	LOCAL CONST Robtarget Tr_meulage_bavure_P268 :=[[-161.9653125,-184.567296875,19.5],[0.560964234006759,-0.570777278642454,0.427648680140188,-0.420296362969132],[0,0,0,0],[8.999999E+09,8.999999E+09,8.999999E+09,8.999999E+09,8.999999E+09,8.999999E+09]];
	LOCAL CONST Robtarget Tr_meulage_bavure_P269 :=[[-161.438453125,-185.88871875,19.5],[0.561482497351615,-0.570629960328972,0.427154440312253,-0.420306956478566],[0,0,0,0],[8.999999E+09,8.999999E+09,8.999999E+09,8.999999E+09,8.999999E+09,8.999999E+09]];
	LOCAL CONST Robtarget Tr_meulage_bavure_P270 :=[[-161.127265625,-186.709515625,19.5],[0.562125073730672,-0.570599348324866,0.426494180054633,-0.420160088007001],[0,0,0,0],[8.999999E+09,8.999999E+09,8.999999E+09,8.999999E+09,8.999999E+09,8.999999E+09]];
	LOCAL CONST Robtarget Tr_meulage_bavure_P271 :=[[-159.300578125,-195.6424375,19.5],[0.562874001364667,-0.570656851193447,0.425695264639237,-0.41988945978369],[0,0,0,0],[8.999999E+09,8.999999E+09,8.999999E+09,8.999999E+09,8.999999E+09,8.999999E+09]];
	LOCAL CONST Robtarget Tr_meulage_bavure_P272 :=[[-159.28934375,-195.682734375,19.5],[0.563712315179465,-0.570787324955456,0.424779737224237,-0.419514517304122],[0,0,0,0],[8.999999E+09,8.999999E+09,8.999999E+09,8.999999E+09,8.999999E+09,8.999999E+09]];
	LOCAL CONST Robtarget Tr_meulage_bavure_P273 :=[[-159.286125,-195.694703125,19.5],[0.564604788725629,-0.570963377966838,0.423792547953419,-0.419072940987527],[0,0,0,0],[8.999999E+09,8.999999E+09,8.999999E+09,8.999999E+09,8.999999E+09,8.999999E+09]];
	LOCAL CONST Robtarget Tr_meulage_bavure_P274 :=[[-159.284375,-195.70196875,19.5],[0.565530486147354,-0.571160305808485,0.422763052996336,-0.418595957132785],[0,0,0,0],[8.999999E+09,8.999999E+09,8.999999E+09,8.999999E+09,8.999999E+09,8.999999E+09]];
	LOCAL CONST Robtarget Tr_meulage_bavure_P275 :=[[-157.99475,-199.292578125,19.5],[0.566472293460366,-0.571359278782923,0.421714944239663,-0.418107906042624],[0,0,0,0],[8.999999E+09,8.999999E+09,8.999999E+09,8.999999E+09,8.999999E+09,8.999999E+09]];
	LOCAL CONST Robtarget Tr_meulage_bavure_P276 :=[[-157.544234375,-200.938265625,19.5],[0.567401299111796,-0.571538107883857,0.420685514492802,-0.417640581000833],[0,0,0,0],[8.999999E+09,8.999999E+09,8.999999E+09,8.999999E+09,8.999999E+09,8.999999E+09]];
	LOCAL CONST Robtarget Tr_meulage_bavure_P277 :=[[-156.8125,-202.558203125,19.5],[0.568302601605658,-0.571679624762868,0.419695994543555,-0.41721676836307],[0,0,0,0],[8.999999E+09,8.999999E+09,8.999999E+09,8.999999E+09,8.999999E+09,8.999999E+09]];
	LOCAL CONST Robtarget Tr_meulage_bavure_P278 :=[[-156.25728125,-204.908390625,19.5],[0.569171214806915,-0.571775396245421,0.418754532827547,-0.416847293046261],[0,0,0,0],[8.999999E+09,8.999999E+09,8.999999E+09,8.999999E+09,8.999999E+09,8.999999E+09]];
	LOCAL CONST Robtarget Tr_meulage_bavure_P279 :=[[-155.75175,-206.384375,19.5],[0.569996546823764,-0.57181706101586,0.417875161306644,-0.416544757382824],[0,0,0,0],[8.999999E+09,8.999999E+09,8.999999E+09,8.999999E+09,8.999999E+09,8.999999E+09]];
	LOCAL CONST Robtarget Tr_meulage_bavure_P280 :=[[-155.11828125,-208.979578125,19.5],[0.570780006509268,-0.571805632479948,0.417056295855806,-0.416308237872519],[0,0,0,0],[8.999999E+09,8.999999E+09,8.999999E+09,8.999999E+09,8.999999E+09,8.999999E+09]];
	LOCAL CONST Robtarget Tr_meulage_bavure_P281 :=[[-154.511328125,-211.640203125,19.5],[0.571520591827226,-0.571739384929797,0.4162997144144,-0.416140404930889],[0,0,0,0],[8.999999E+09,8.999999E+09,8.999999E+09,8.999999E+09,8.999999E+09,8.999999E+09]];
	LOCAL CONST Robtarget Tr_meulage_bavure_P282 :=[[-154.18290625,-212.67675,19.5],[0.572213364310843,-0.57162923861389,0.415607199226649,-0.416031892066882],[0,0,0,0],[8.999999E+09,8.999999E+09,8.999999E+09,8.999999E+09,8.999999E+09,8.999999E+09]];
	LOCAL CONST Robtarget Tr_meulage_bavure_P283 :=[[-152.8583125,-215.9785,19.5],[0.572864706832717,-0.571464182646808,0.414975670626358,-0.415992678307547],[0,0,0,0],[8.999999E+09,8.999999E+09,8.999999E+09,8.999999E+09,8.999999E+09,8.999999E+09]];
	LOCAL CONST Robtarget Tr_meulage_bavure_P284 :=[[-152.411953125,-217.957359375,19.5],[0.573480034959651,-0.571248401283081,0.4143980984857,-0.416016982232263],[0,0,0,0],[8.999999E+09,8.999999E+09,8.999999E+09,8.999999E+09,8.999999E+09,8.999999E+09]];
	LOCAL CONST Robtarget Tr_meulage_bavure_P285 :=[[-151.933640625,-219.27084375,19.5],[0.574050202363302,-0.570970854337552,0.413887624220456,-0.416119794267042],[0,0,0,0],[8.999999E+09,8.999999E+09,8.999999E+09,8.999999E+09,8.999999E+09,8.999999E+09]];
	LOCAL CONST Robtarget Tr_meulage_bavure_P286 :=[[-151.668234375,-220.093296875,19.5],[0.574574547686089,-0.570649212284852,0.413439168547303,-0.416283100282631],[0,0,0,0],[8.999999E+09,8.999999E+09,8.999999E+09,8.999999E+09,8.999999E+09,8.999999E+09]];
	LOCAL CONST Robtarget Tr_meulage_bavure_P287 :=[[-149.616609375,-228.880140625,19.5],[0.575057843902687,-0.570279616930627,0.413048830883079,-0.41650966133521],[0,0,0,0],[8.999999E+09,8.999999E+09,8.999999E+09,8.999999E+09,8.999999E+09,8.999999E+09]];
	LOCAL CONST Robtarget Tr_meulage_bavure_P288 :=[[-149.551046875,-229.11575,19.5],[0.575509045661707,-0.569878410393925,0.412701822474269,-0.416779487804835],[0,0,0,0],[8.999999E+09,8.999999E+09,8.999999E+09,8.999999E+09,8.999999E+09,8.999999E+09]];
	LOCAL CONST Robtarget Tr_meulage_bavure_P289 :=[[-147.845921875,-233.037921875,19.5],[0.575938029590918,-0.569448353003208,0.412386744830926,-0.417086480265925],[0,0,0,0],[8.999999E+09,8.999999E+09,8.999999E+09,8.999999E+09,8.999999E+09,8.999999E+09]];
	LOCAL CONST Robtarget Tr_meulage_bavure_P290 :=[[-147.505546875,-234.7584375,19.5],[0.576374910636539,-0.569018116570961,0.412062744044535,-0.417390273453091],[0,0,0,0],[8.999999E+09,8.999999E+09,8.999999E+09,8.999999E+09,8.999999E+09,8.999999E+09]];
	LOCAL CONST Robtarget Tr_meulage_bavure_P291 :=[[-146.999359375,-236.0205,19.5],[0.576853982153147,-0.568620156737828,0.411683557372683,-0.417644884099493],[0,0,0,0],[8.999999E+09,8.999999E+09,8.999999E+09,8.999999E+09,8.999999E+09,8.999999E+09]];
	LOCAL CONST Robtarget Tr_meulage_bavure_P292 :=[[-146.427,-238.509484375,19.5],[0.577416776077298,-0.568301736935537,0.41119083020271,-0.417785954356722],[0,0,0,0],[8.999999E+09,8.999999E+09,8.999999E+09,8.999999E+09,8.999999E+09,8.999999E+09]];
	LOCAL CONST Robtarget Tr_meulage_bavure_P293 :=[[-146.179640625,-239.26884375,19.5],[0.578126284754704,-0.568116391381928,0.410501698615583,-0.417734509171339],[0,0,0,0],[8.999999E+09,8.999999E+09,8.999999E+09,8.999999E+09,8.999999E+09,8.999999E+09]];
	LOCAL CONST Robtarget Tr_meulage_bavure_P294 :=[[-145.538734375,-242.18440625,19.5],[0.57903388760407,-0.568130354419907,0.409541192289515,-0.417401089134791],[0,0,0,0],[8.999999E+09,8.999999E+09,8.999999E+09,8.999999E+09,8.999999E+09,8.999999E+09]];
	LOCAL CONST Robtarget Tr_meulage_bavure_P295 :=[[-145.2123125,-243.432875,19.5],[0.580214944471463,-0.568413693302016,0.408206746970448,-0.416681824905458],[0,0,0,0],[8.999999E+09,8.999999E+09,8.999999E+09,8.999999E+09,8.999999E+09,8.999999E+09]];
	LOCAL CONST Robtarget Tr_meulage_bavure_P296 :=[[-144.365421875,-245.033828125,19.5],[0.581756623872827,-0.569033712901752,0.406381818028901,-0.415468027815452],[0,0,0,0],[8.999999E+09,8.999999E+09,8.999999E+09,8.999999E+09,8.999999E+09,8.999999E+09]];
	LOCAL CONST Robtarget Tr_meulage_bavure_P297 :=[[-144.034125,-246.257625,19.5],[0.583714280713272,-0.570060460460229,0.403978570192655,-0.413654475059025],[0,0,0,0],[8.999999E+09,8.999999E+09,8.999999E+09,8.999999E+09,8.999999E+09,8.999999E+09]];
	LOCAL CONST Robtarget Tr_meulage_bavure_P298 :=[[-143.6095,-247.7546875,19.5],[0.58617245989944,-0.571557348115518,0.400874380777533,-0.4111250125045],[0,0,0,0],[8.999999E+09,8.999999E+09,8.999999E+09,8.999999E+09,8.999999E+09,8.999999E+09]];
	LOCAL CONST Robtarget Tr_meulage_bavure_P299 :=[[-142.860328125,-249.55490625,19.5],[0.589188052385461,-0.573590439879237,0.396966412920798,-0.407761098215811],[0,0,0,0],[8.999999E+09,8.999999E+09,8.999999E+09,8.999999E+09,8.999999E+09,8.999999E+09]];
	LOCAL CONST Robtarget Tr_meulage_bavure_P300 :=[[-142.402375,-251.853640625,19.5],[0.592808671964743,-0.576208210016921,0.392156346958513,-0.403454305581994],[0,0,0,0],[8.999999E+09,8.999999E+09,8.999999E+09,8.999999E+09,8.999999E+09,8.999999E+09]];
	LOCAL CONST Robtarget Tr_meulage_bavure_P301 :=[[-140.7485625,-258.0768125,19.5],[0.597072072972443,-0.579441265135707,0.386348990807515,-0.398104530539827],[0,0,0,0],[8.999999E+09,8.999999E+09,8.999999E+09,8.999999E+09,8.999999E+09,8.999999E+09]];
	LOCAL CONST Robtarget Tr_meulage_bavure_P302 :=[[-140.3933125,-259.20978125,19.5],[0.602013083361173,-0.583316118473957,0.379437191320676,-0.391599248254036],[0,0,0,0],[8.999999E+09,8.999999E+09,8.999999E+09,8.999999E+09,8.999999E+09,8.999999E+09]];
	LOCAL CONST Robtarget Tr_meulage_bavure_P303 :=[[-140.164671875,-259.836421875,19.5],[0.607618116502847,-0.587817465101063,0.371364545167804,-0.383873972563918],[0,0,0,0],[8.999999E+09,8.999999E+09,8.999999E+09,8.999999E+09,8.999999E+09,8.999999E+09]];
	LOCAL CONST Robtarget Tr_meulage_bavure_P304 :=[[-138.449671875,-263.1504375,19.5],[0.613883056235529,-0.592942762212286,0.362039441275421,-0.374825181875461],[0,0,0,0],[8.999999E+09,8.999999E+09,8.999999E+09,8.999999E+09,8.999999E+09,8.999999E+09]];
	LOCAL CONST Robtarget Tr_meulage_bavure_P305 :=[[-137.6564375,-265.19478125,19.5],[0.620753084659352,-0.59864213211971,0.351426859012845,-0.36440687191851],[0,0,0,0],[8.999999E+09,8.999999E+09,8.999999E+09,8.999999E+09,8.999999E+09,8.999999E+09]];
	LOCAL CONST Robtarget Tr_meulage_bavure_P306 :=[[-136.8803125,-266.6085625,19.5],[0.628170166944891,-0.604841141121465,0.339490203423159,-0.35258451064534],[0,0,0,0],[8.999999E+09,8.999999E+09,8.999999E+09,8.999999E+09,8.999999E+09,8.999999E+09]];
	LOCAL CONST Robtarget Tr_meulage_bavure_P307 :=[[-134.9164375,-269.53475,19.5],[0.636031217124536,-0.611449574748402,0.326239235907522,-0.339354783873095],[0,0,0,0],[8.999999E+09,8.999999E+09,8.999999E+09,8.999999E+09,8.999999E+09,8.999999E+09]];
	LOCAL CONST Robtarget Tr_meulage_bavure_P308 :=[[-133.2449375,-272.6095625,19.5],[0.644224659383251,-0.618344665454578,0.311705957595993,-0.32475199606094],[0,0,0,0],[8.999999E+09,8.999999E+09,8.999999E+09,8.999999E+09,8.999999E+09,8.999999E+09]];
	LOCAL CONST Robtarget Tr_meulage_bavure_P309 :=[[-132.551703125,-273.5116875,19.5],[0.652594348190598,-0.625402876804148,0.29598013661176,-0.308848858061784],[0,0,0,0],[8.999999E+09,8.999999E+09,8.999999E+09,8.999999E+09,8.999999E+09,8.999999E+09]];
	LOCAL CONST Robtarget Tr_meulage_bavure_P310 :=[[-132.1574375,-273.93109375,19.5],[0.660998089293367,-0.63246286972877,0.27917792373045,-0.291773767269302],[0,0,0,0],[8.999999E+09,8.999999E+09,8.999999E+09,8.999999E+09,8.999999E+09,8.999999E+09]];
	LOCAL CONST Robtarget Tr_meulage_bavure_P311 :=[[-130.1533828125,-275.91075,19.5],[0.669271343454706,-0.639374635521518,0.261469816707866,-0.273695961301611],[0,0,0,0],[8.999999E+09,8.999999E+09,8.999999E+09,8.999999E+09,8.999999E+09,8.999999E+09]];
	LOCAL CONST Robtarget Tr_meulage_bavure_P312 :=[[-129.5635390625,-276.394625,19.5],[0.677256054189009,-0.645991723265792,0.243065647445525,-0.25482939698613],[0,0,0,0],[8.999999E+09,8.999999E+09,8.999999E+09,8.999999E+09,8.999999E+09,8.999999E+09]];
	LOCAL CONST Robtarget Tr_meulage_bavure_P313 :=[[-125.70825,-279.1965,19.5],[0.684815904495517,-0.652189819896316,0.224188779708599,-0.235403922708113],[0,0,0,0],[8.999999E+09,8.999999E+09,8.999999E+09,8.999999E+09,8.999999E+09,8.999999E+09]];
	LOCAL CONST Robtarget Tr_meulage_bavure_P314 :=[[-124.69521875,-279.913875,19.5],[0.691839849635144,-0.657856194737078,0.205091279018427,-0.215685921593087],[0,0,0,0],[8.999999E+09,8.999999E+09,8.999999E+09,8.999999E+09,8.999999E+09,8.999999E+09]];
	LOCAL CONST Robtarget Tr_meulage_bavure_P315 :=[[-119.5407109375,-282.797625,19.5],[0.698244372547129,-0.662926894954686,0.186008064006495,-0.195917656877987],[0,0,0,0],[8.999999E+09,8.999999E+09,8.999999E+09,8.999999E+09,8.999999E+09,8.999999E+09]];
	LOCAL CONST Robtarget Tr_meulage_bavure_P316 :=[[-116.7555546875,-284.14571875,19.5],[0.703994145177397,-0.667352092209407,0.167154061077636,-0.176331926901872],[0,0,0,0],[8.999999E+09,8.999999E+09,8.999999E+09,8.999999E+09,8.999999E+09,8.999999E+09]];
	LOCAL CONST Robtarget Tr_meulage_bavure_P317 :=[[-112.591765625,-285.93153125,19.5],[0.709058736177083,-0.67112758152923,0.148747698148336,-0.157154701670856],[0,0,0,0],[8.999999E+09,8.999999E+09,8.999999E+09,8.999999E+09,8.999999E+09,8.999999E+09]];
	LOCAL CONST Robtarget Tr_meulage_bavure_P318 :=[[-111.89978125,-286.17246875,19.5],[0.713459335022752,-0.674262369715255,0.130947400243534,-0.138559779244634],[0,0,0,0],[8.999999E+09,8.999999E+09,8.999999E+09,8.999999E+09,8.999999E+09,8.999999E+09]];
	LOCAL CONST Robtarget Tr_meulage_bavure_P319 :=[[-109.451328125,-286.99928125,19.5],[0.71721616316262,-0.676798706879172,0.113904788557829,-0.120707020543821],[0,0,0,0],[8.999999E+09,8.999999E+09,8.999999E+09,8.999999E+09,8.999999E+09,8.999999E+09]];
	LOCAL CONST Robtarget Tr_meulage_bavure_P320 :=[[-109.0068671875,-287.11028125,19.5],[0.720386199432233,-0.678781129299869,0.0977080074532281,-0.103696901851012],[0,0,0,0],[8.999999E+09,8.999999E+09,8.999999E+09,8.999999E+09,8.999999E+09,8.999999E+09]];
	LOCAL CONST Robtarget Tr_meulage_bavure_P321 :=[[-107.78265625,-287.435875,19.5],[0.723031240066771,-0.680253807562518,0.0824577376474849,-0.0876430526982125],[0,0,0,0],[8.999999E+09,8.999999E+09,8.999999E+09,8.999999E+09,8.999999E+09,8.999999E+09]];
	LOCAL CONST Robtarget Tr_meulage_bavure_P322 :=[[-106.4644453125,-287.84596875,19.5],[0.7252109507937,-0.681285287306183,0.0681925909536574,-0.0725892876949244],[0,0,0,0],[8.999999E+09,8.999999E+09,8.999999E+09,8.999999E+09,8.999999E+09,8.999999E+09]];
	LOCAL CONST Robtarget Tr_meulage_bavure_P323 :=[[-105.98046875,-287.92040625,19.5],[0.726986745083191,-0.681934622504451,0.0549682733471719,-0.0585997613330488],[0,0,0,0],[8.999999E+09,8.999999E+09,8.999999E+09,8.999999E+09,8.999999E+09,8.999999E+09]];
	LOCAL CONST Robtarget Tr_meulage_bavure_P324 :=[[-105.7509140625,-287.94509375,19.5],[0.728412623159497,-0.682271282005315,0.0428061076178847,-0.0457010429129395],[0,0,0,0],[8.999999E+09,8.999999E+09,8.999999E+09,8.999999E+09,8.999999E+09,8.999999E+09]];
	LOCAL CONST Robtarget Tr_meulage_bavure_P325 :=[[-103.7956875,-287.85703125,19.5],[0.729555020391346,-0.682343993654236,0.0317183960258636,-0.0339129753828471],[0,0,0,0],[8.999999E+09,8.999999E+09,8.999999E+09,8.999999E+09,8.999999E+09,8.999999E+09]];
	LOCAL CONST Robtarget Tr_meulage_bavure_P326 :=[[-98.836609375,-287.8770625,19.5],[0.730465389526081,-0.682208988231543,0.0217049125177494,-0.0232402205928225],[0,0,0,0],[8.999999E+09,8.999999E+09,8.999999E+09,8.999999E+09,8.999999E+09,8.999999E+09]];
	LOCAL CONST Robtarget Tr_meulage_bavure_P327 :=[[-98.1267734375,-287.92809375,19.5],[0.731193592992967,-0.681913551506533,0.0127567102372147,-0.013678603061212],[0,0,0,0],[8.999999E+09,8.999999E+09,8.999999E+09,8.999999E+09,8.999999E+09,8.999999E+09]];
	LOCAL CONST Robtarget Tr_meulage_bavure_P328 :=[[-96.89046875,-287.7645625,19.5],[0.731783571389712,-0.681499822687102,0.00485727743171576,-0.00521566654587902],[0,0,0,0],[8.999999E+09,8.999999E+09,8.999999E+09,8.999999E+09,8.999999E+09,8.999999E+09]];
	LOCAL CONST Robtarget Tr_meulage_bavure_P329 :=[[-95.0238984375,-287.6898125,19.5],[0.732277533985066,-0.680999874855432,-0.00201830542058397,0.00217027898357202],[0,0,0,0],[8.999999E+09,8.999999E+09,8.999999E+09,8.999999E+09,8.999999E+09,8.999999E+09]];
	LOCAL CONST Robtarget Tr_meulage_bavure_P330 :=[[-91.72903125,-287.34909375,19.5],[0.732701770281004,-0.680451088617369,-0.0078900027828738,0.00849586267586157],[0,0,0,0],[8.999999E+09,8.999999E+09,8.999999E+09,8.999999E+09,8.999999E+09,8.999999E+09]];
	LOCAL CONST Robtarget Tr_meulage_bavure_P331 :=[[-89.856875,-287.0336875,19.5],[0.733088866138208,-0.679871664260582,-0.0128162700320661,0.0138194682317681],[0,0,0,0],[8.999999E+09,8.999999E+09,8.999999E+09,8.999999E+09,8.999999E+09,8.999999E+09]];
	LOCAL CONST Robtarget Tr_meulage_bavure_P332 :=[[-85.5172734375,-286.69559375,19.5],[0.733453444169888,-0.67928812631057,-0.0168329671656543,0.0181752002795984],[0,0,0,0],[8.999999E+09,8.999999E+09,8.999999E+09,8.999999E+09,8.999999E+09,8.999999E+09]];
	LOCAL CONST Robtarget Tr_meulage_bavure_P333 :=[[-84.53634375,-286.54434375,19.5],[0.733821815164145,-0.678703060287681,-0.0200010590824421,0.0216253827923831],[0,0,0,0],[8.999999E+09,8.999999E+09,8.999999E+09,8.999999E+09,8.999999E+09,8.999999E+09]];
	LOCAL CONST Robtarget Tr_meulage_bavure_P334 :=[[-83.2665078125,-286.44875,19.5],[0.734198119116665,-0.678132647710818,-0.0223929803954049,0.0242443482749612],[0,0,0,0],[8.999999E+09,8.999999E+09,8.999999E+09,8.999999E+09,8.999999E+09,8.999999E+09]];
	LOCAL CONST Robtarget Tr_meulage_bavure_P335 :=[[-79.6076640625,-285.996375,19.5],[0.734583912009596,-0.677588173949316,-0.0240742626965029,0.0260992838279178],[0,0,0,0],[8.999999E+09,8.999999E+09,8.999999E+09,8.999999E+09,8.999999E+09,8.999999E+09]];
	LOCAL CONST Robtarget Tr_meulage_bavure_P336 :=[[-78.2538125,-285.63596875,19.5],[0.734986132932684,-0.67706581152781,-0.0251443204817685,0.0272953183596925],[0,0,0,0],[8.999999E+09,8.999999E+09,8.999999E+09,8.999999E+09,8.999999E+09,8.999999E+09]];
	LOCAL CONST Robtarget Tr_meulage_bavure_P337 :=[[-76.3402109375,-285.37465625,19.5],[0.735402485292143,-0.676567290093219,-0.0256914156380045,0.0279255754564468],[0,0,0,0],[8.999999E+09,8.999999E+09,8.999999E+09,8.999999E+09,8.999999E+09,8.999999E+09]];
	LOCAL CONST Robtarget Tr_meulage_bavure_P338 :=[[-72.4418359375,-285.24371875,19.5],[0.735825551022483,-0.67609503373989,-0.0258192860533249,0.0281003253079716],[0,0,0,0],[8.999999E+09,8.999999E+09,8.999999E+09,8.999999E+09,8.999999E+09,8.999999E+09]];
	LOCAL CONST Robtarget Tr_meulage_bavure_P339 :=[[-68.4656953125,-284.83971875,19.5],[0.736267597026046,-0.675628090950229,-0.0256273793944011,0.0279275081920483],[0,0,0,0],[8.999999E+09,8.999999E+09,8.999999E+09,8.999999E+09,8.999999E+09,8.999999E+09]];
	LOCAL CONST Robtarget Tr_meulage_bavure_P340 :=[[-65.6481015625,-284.45584375,19.5],[0.736706993967259,-0.675179101732153,-0.0252442696560809,0.0275447358567801],[0,0,0,0],[8.999999E+09,8.999999E+09,8.999999E+09,8.999999E+09,8.999999E+09,8.999999E+09]];
	LOCAL CONST Robtarget Tr_meulage_bavure_P341 :=[[-64.50961328125,-284.47453125,19.5],[0.737145027213847,-0.674739001078387,-0.0247574912343207,0.0270472901677574],[0,0,0,0],[8.999999E+09,8.999999E+09,8.999999E+09,8.999999E+09,8.999999E+09,8.999999E+09]];
	LOCAL CONST Robtarget Tr_meulage_bavure_P342 :=[[-63.09558203125,-284.451,19.5],[0.737574727550139,-0.674306700194866,-0.0242719686569887,0.0265493293542989],[0,0,0,0],[8.999999E+09,8.999999E+09,8.999999E+09,8.999999E+09,8.999999E+09,8.999999E+09]];
	LOCAL CONST Robtarget Tr_meulage_bavure_P343 :=[[-60.75375390625,-284.1825,19.5],[0.737995519441899,-0.673876223593398,-0.0238729311077847,0.0261444395523303],[0,0,0,0],[8.999999E+09,8.999999E+09,8.999999E+09,8.999999E+09,8.999999E+09,8.999999E+09]];
	LOCAL CONST Robtarget Tr_meulage_bavure_P344 :=[[-56.9111328125,-283.74796875,19.5],[0.738407827244645,-0.673441766800905,-0.0236337028553787,0.0259136157504544],[0,0,0,0],[8.999999E+09,8.999999E+09,8.999999E+09,8.999999E+09,8.999999E+09,8.999999E+09]];
	LOCAL CONST Robtarget Tr_meulage_bavure_P345 :=[[-55.53506640625,-283.48496875,19.5],[0.738803521845753,-0.673007813207025,-0.0236162827783587,0.0259250970748975],[0,0,0,0],[8.999999E+09,8.999999E+09,8.999999E+09,8.999999E+09,8.999999E+09,8.999999E+09]];
	LOCAL CONST Robtarget Tr_meulage_bavure_P346 :=[[-53.50186328125,-283.17409375,19.5],[0.739190986070497,-0.672563047793711,-0.0238471875011445,0.0262096261485151],[0,0,0,0],[8.999999E+09,8.999999E+09,8.999999E+09,8.999999E+09,8.999999E+09,8.999999E+09]];
	LOCAL CONST Robtarget Tr_meulage_bavure_P347 :=[[-49.17727734375,-282.77846875,19.5],[0.739554654010651,-0.672122706016185,-0.0243425371632662,0.0267847470236889],[0,0,0,0],[8.999999E+09,8.999999E+09,8.999999E+09,8.999999E+09,8.999999E+09,8.999999E+09]];
	LOCAL CONST Robtarget Tr_meulage_bavure_P348 :=[[-44.38299609375,-282.44271875,19.5],[0.739908728288621,-0.671670717382305,-0.0250908871651308,0.0276399818148069],[0,0,0,0],[8.999999E+09,8.999999E+09,8.999999E+09,8.999999E+09,8.999999E+09,8.999999E+09]];
	LOCAL CONST Robtarget Tr_meulage_bavure_P349 :=[[-41.2405390625,-282.2865,19.5],[0.740250211472266,-0.671209902210246,-0.0260751504918529,0.0287572272134317],[0,0,0,0],[8.999999E+09,8.999999E+09,8.999999E+09,8.999999E+09,8.999999E+09,8.999999E+09]];
	LOCAL CONST Robtarget Tr_meulage_bavure_P350 :=[[-37.7456953125,-282.0811875,19.5],[0.740566887367051,-0.670755399045768,-0.0272511663274277,0.0300874379139331],[0,0,0,0],[8.999999E+09,8.999999E+09,8.999999E+09,8.999999E+09,8.999999E+09,8.999999E+09]];
	LOCAL CONST Robtarget Tr_meulage_bavure_P351 :=[[-35.7432265625,-281.81509375,19.5],[0.740869701006427,-0.670297395744423,-0.0285705731810239,0.0315786278517456],[0,0,0,0],[8.999999E+09,8.999999E+09,8.999999E+09,8.999999E+09,8.999999E+09,8.999999E+09]];
	LOCAL CONST Robtarget Tr_meulage_bavure_P352 :=[[-32.817078125,-281.2908125,19.5],[0.741163425883474,-0.669833608837101,-0.0299837116955564,0.0331766429569906],[0,0,0,0],[8.999999E+09,8.999999E+09,8.999999E+09,8.999999E+09,8.999999E+09,8.999999E+09]];
	LOCAL CONST Robtarget Tr_meulage_bavure_P353 :=[[-31.189666015625,-281.02409375,19.5],[0.741439666191449,-0.669378732229863,-0.0314264722459313,0.0348096405961052],[0,0,0,0],[8.999999E+09,8.999999E+09,8.999999E+09,8.999999E+09,8.999999E+09,8.999999E+09]];
	LOCAL CONST Robtarget Tr_meulage_bavure_P354 :=[[-28.535064453125,-280.90421875,19.5],[0.741714526644082,-0.668919898476124,-0.0328488839806384,0.0364236353081897],[0,0,0,0],[8.999999E+09,8.999999E+09,8.999999E+09,8.999999E+09,8.999999E+09,8.999999E+09]];
	LOCAL CONST Robtarget Tr_meulage_bavure_P355 :=[[-23.35043359375,-280.3699375,19.5],[0.741979260892866,-0.668474452748739,-0.0341871288687678,0.0379463126912225],[0,0,0,0],[8.999999E+09,8.999999E+09,8.999999E+09,8.999999E+09,8.999999E+09,8.999999E+09]];
	LOCAL CONST Robtarget Tr_meulage_bavure_P356 :=[[-21.707732421875,-280.1441875,19.5],[0.742239132342601,-0.668041110268359,-0.0354126033921952,0.0393458121241323],[0,0,0,0],[8.999999E+09,8.999999E+09,8.999999E+09,8.999999E+09,8.999999E+09,8.999999E+09]];
	LOCAL CONST Robtarget Tr_meulage_bavure_P357 :=[[-18.087798828125,-279.7083125,19.5],[0.742510743010949,-0.667607685693368,-0.0364850387971614,0.0405785221569577],[0,0,0,0],[8.999999E+09,8.999999E+09,8.999999E+09,8.999999E+09,8.999999E+09,8.999999E+09]];
	LOCAL CONST Robtarget Tr_meulage_bavure_P358 :=[[-17.23358203125,-279.54203125,19.5],[0.742787417657644,-0.667185113955726,-0.0373904077498098,0.0416273142741171],[0,0,0,0],[8.999999E+09,8.999999E+09,8.999999E+09,8.999999E+09,8.999999E+09,8.999999E+09]];
	LOCAL CONST Robtarget Tr_meulage_bavure_P359 :=[[-15.7358095703125,-279.48275,19.5],[0.743060843326873,-0.666786518977901,-0.038111731974697,0.0424713681152043],[0,0,0,0],[8.999999E+09,8.999999E+09,8.999999E+09,8.999999E+09,8.999999E+09,8.999999E+09]];
	LOCAL CONST Robtarget Tr_meulage_bavure_P360 :=[[-11.11053515625,-278.86453125,19.5],[0.74334126114516,-0.66640177114528,-0.0386497263769758,0.0431120347993692],[0,0,0,0],[8.999999E+09,8.999999E+09,8.999999E+09,8.999999E+09,8.999999E+09,8.999999E+09]];
	LOCAL CONST Robtarget Tr_meulage_bavure_P361 :=[[-9.1521298828125,-278.51259375,19.5],[0.743625034281882,-0.666035033451219,-0.0390121073460656,0.0435568374118436],[0,0,0,0],[8.999999E+09,8.999999E+09,8.999999E+09,8.999999E+09,8.999999E+09,8.999999E+09]];
	LOCAL CONST Robtarget Tr_meulage_bavure_P362 :=[[-4.1391904296875,-278.02171875,19.5],[0.743913750798036,-0.665683653011691,-0.0392109822866391,0.043818995364179],[0,0,0,0],[8.999999E+09,8.999999E+09,8.999999E+09,8.999999E+09,8.999999E+09,8.999999E+09]];
	LOCAL CONST Robtarget Tr_meulage_bavure_P363 :=[[3.73715209960938,-277.50453125,19.5],[0.744208876706379,-0.665343612809414,-0.0392671951058527,0.0439216588218871],[0,0,0,0],[8.999999E+09,8.999999E+09,8.999999E+09,8.999999E+09,8.999999E+09,8.999999E+09]];
	LOCAL CONST Robtarget Tr_meulage_bavure_P364 :=[[4.41998291015625,-277.3703125,19.5],[0.744509424422736,-0.665014123771272,-0.0391961306942008,0.0438816074119574],[0,0,0,0],[8.999999E+09,8.999999E+09,8.999999E+09,8.999999E+09,8.999999E+09,8.999999E+09]];
	LOCAL CONST Robtarget Tr_meulage_bavure_P365 :=[[6.283447265625,-277.18909375,19.5],[0.744804935293087,-0.664703307286453,-0.0390252875238091,0.0437281211487018],[0,0,0,0],[8.999999E+09,8.999999E+09,8.999999E+09,8.999999E+09,8.999999E+09,8.999999E+09]];
	LOCAL CONST Robtarget Tr_meulage_bavure_P366 :=[[14.9065546875,-276.00421875,19.5],[0.745101806435219,-0.664401693705879,-0.0387708064935192,0.0434800185323727],[0,0,0,0],[8.999999E+09,8.999999E+09,8.999999E+09,8.999999E+09,8.999999E+09,8.999999E+09]];
	LOCAL CONST Robtarget Tr_meulage_bavure_P367 :=[[17.427978515625,-275.71321875,19.5],[0.745395572448328,-0.664111310053286,-0.0384543515048626,0.0431609926215477],[0,0,0,0],[8.999999E+09,8.999999E+09,8.999999E+09,8.999999E+09,8.999999E+09,8.999999E+09]];
	LOCAL CONST Robtarget Tr_meulage_bavure_P368 :=[[22.690033203125,-274.89740625,19.5],[0.745689508202804,-0.663825992976087,-0.0380935305284928,0.0427912530483325],[0,0,0,0],[8.999999E+09,8.999999E+09,8.999999E+09,8.999999E+09,8.999999E+09,8.999999E+09]];
	LOCAL CONST Robtarget Tr_meulage_bavure_P369 :=[[24.436462890625,-274.65103125,19.5],[0.745982896599928,-0.663544527508919,-0.0377029252851454,0.0423871138235338],[0,0,0,0],[8.999999E+09,8.999999E+09,8.999999E+09,8.999999E+09,8.999999E+09,8.999999E+09]];
	LOCAL CONST Robtarget Tr_meulage_bavure_P370 :=[[27.416291015625,-274.272,19.5],[0.746268856927678,-0.663272002159742,-0.0373028883472666,0.0419706903900203],[0,0,0,0],[8.999999E+09,8.999999E+09,8.999999E+09,8.999999E+09,8.999999E+09,8.999999E+09]];
	LOCAL CONST Robtarget Tr_meulage_bavure_P371 :=[[28.458375,-274.05478125,19.5],[0.746550366383039,-0.663004858448019,-0.0368947035688752,0.0415438199524097],[0,0,0,0],[8.999999E+09,8.999999E+09,8.999999E+09,8.999999E+09,8.999999E+09,8.999999E+09]];
	LOCAL CONST Robtarget Tr_meulage_bavure_P372 :=[[30.38855078125,-273.92025,19.5],[0.746830255296542,-0.662736357267652,-0.0365063043339479,0.0411385497214313],[0,0,0,0],[8.999999E+09,8.999999E+09,8.999999E+09,8.999999E+09,8.999999E+09,8.999999E+09]];
	LOCAL CONST Robtarget Tr_meulage_bavure_P373 :=[[33.11441015625,-273.5259375,19.5],[0.747099570603815,-0.662477919835629,-0.0361281719578439,0.0407430058395047],[0,0,0,0],[8.999999E+09,8.999999E+09,8.999999E+09,8.999999E+09,8.999999E+09,8.999999E+09]];
	LOCAL CONST Robtarget Tr_meulage_bavure_P374 :=[[34.83148046875,-273.24446875,19.5],[0.747355157433442,-0.662229707584567,-0.0357885259274169,0.0403889150886211],[0,0,0,0],[8.999999E+09,8.999999E+09,8.999999E+09,8.999999E+09,8.999999E+09,8.999999E+09]];
	LOCAL CONST Robtarget Tr_meulage_bavure_P375 :=[[38.11590625,-272.91428125,19.5],[0.747610535984406,-0.66197542874325,-0.0354960931727873,0.0400879731935678],[0,0,0,0],[8.999999E+09,8.999999E+09,8.999999E+09,8.999999E+09,8.999999E+09,8.999999E+09]];
	LOCAL CONST Robtarget Tr_meulage_bavure_P376 :=[[39.43502734375,-272.83925,19.5],[0.747850297504655,-0.661731773858748,-0.0352587508784534,0.0398473647114343],[0,0,0,0],[8.999999E+09,8.999999E+09,8.999999E+09,8.999999E+09,8.999999E+09,8.999999E+09]];
	LOCAL CONST Robtarget Tr_meulage_bavure_P377 :=[[45.2320859375,-272.17715625,19.5],[0.748080186236866,-0.661490302975661,-0.0350933746847424,0.0396871400105893],[0,0,0,0],[8.999999E+09,8.999999E+09,8.999999E+09,8.999999E+09,8.999999E+09,8.999999E+09]];
	LOCAL CONST Robtarget Tr_meulage_bavure_P378 :=[[47.62060546875,-271.8248125,19.5],[0.748297266506116,-0.661254439010767,-0.0350002595066617,0.0396074445337873],[0,0,0,0],[8.999999E+09,8.999999E+09,8.999999E+09,8.999999E+09,8.999999E+09,8.999999E+09]];
	LOCAL CONST Robtarget Tr_meulage_bavure_P379 :=[[48.34982421875,-271.83715625,19.5],[0.748503119203697,-0.661021600007927,-0.0349864096413146,0.039616612749036],[0,0,0,0],[8.999999E+09,8.999999E+09,8.999999E+09,8.999999E+09,8.999999E+09,8.999999E+09]];
	LOCAL CONST Robtarget Tr_meulage_bavure_P380 :=[[52.699859375,-271.37153125,19.5],[0.748708790454047,-0.660778572494331,-0.0350569386395885,0.0397219873925214],[0,0,0,0],[8.999999E+09,8.999999E+09,8.999999E+09,8.999999E+09,8.999999E+09,8.999999E+09]];
	LOCAL CONST Robtarget Tr_meulage_bavure_P381 :=[[54.4260546875,-271.0833125,19.5],[0.748899486297266,-0.660541882838812,-0.0352139747839537,0.0399243837693531],[0,0,0,0],[8.999999E+09,8.999999E+09,8.999999E+09,8.999999E+09,8.999999E+09,8.999999E+09]];
	LOCAL CONST Robtarget Tr_meulage_bavure_P382 :=[[55.685546875,-271.07,19.5],[0.749080580145308,-0.660306485593583,-0.0354475195835911,0.0402132178219008],[0,0,0,0],[8.999999E+09,8.999999E+09,8.999999E+09,8.999999E+09,8.999999E+09,8.999999E+09]];
	LOCAL CONST Robtarget Tr_meulage_bavure_P383 :=[[61.25250390625,-270.677625,19.5],[0.749249993862185,-0.660071830983981,-0.0357795012722655,0.0406134451589521],[0,0,0,0],[8.999999E+09,8.999999E+09,8.999999E+09,8.999999E+09,8.999999E+09,8.999999E+09]];
	LOCAL CONST Robtarget Tr_meulage_bavure_P384 :=[[61.646484375,-270.614125,19.5],[0.749411887250001,-0.659833714763356,-0.0362027313846949,0.0411175674167231],[0,0,0,0],[8.999999E+09,8.999999E+09,8.999999E+09,8.999999E+09,8.999999E+09,8.999999E+09]];
	LOCAL CONST Robtarget Tr_meulage_bavure_P385 :=[[61.9664296875,-270.596875,19.5],[0.749555868186807,-0.659601425194716,-0.036734234496255,0.0417439380484813],[0,0,0,0],[8.999999E+09,8.999999E+09,8.999999E+09,8.999999E+09,8.999999E+09,8.999999E+09]];
	LOCAL CONST Robtarget Tr_meulage_bavure_P386 :=[[67.4912421875,-269.82709375,19.5],[0.749684084891055,-0.659367738775831,-0.0374058686854177,0.0425295063526245],[0,0,0,0],[8.999999E+09,8.999999E+09,8.999999E+09,8.999999E+09,8.999999E+09,8.999999E+09]];
	LOCAL CONST Robtarget Tr_meulage_bavure_P387 :=[[69.15759375,-269.49821875,19.5],[0.749800250470714,-0.659124792175536,-0.0382370814766123,0.0434973370881756],[0,0,0,0],[8.999999E+09,8.999999E+09,8.999999E+09,8.999999E+09,8.999999E+09,8.999999E+09]];
	LOCAL CONST Robtarget Tr_meulage_bavure_P388 :=[[72.301265625,-268.82734375,19.5],[0.74988567242769,-0.658884441579498,-0.0392872343814879,0.0447133553516025],[0,0,0,0],[8.999999E+09,8.999999E+09,8.999999E+09,8.999999E+09,8.999999E+09,8.999999E+09]];
	LOCAL CONST Robtarget Tr_meulage_bavure_P389 :=[[209.292484375,-254.7383125,19.5],[0.749950261226932,-0.658625066039587,-0.0406112121990249,0.0462423778987642],[0,0,0,0],[8.999999E+09,8.999999E+09,8.999999E+09,8.999999E+09,8.999999E+09,8.999999E+09]];
	LOCAL CONST Robtarget Tr_meulage_bavure_P390 :=[[209.595640625,-254.598515625,19.5],[0.749979833975741,-0.658348824535315,-0.0422781521533605,0.0481625550940398],[0,0,0,0],[8.999999E+09,8.999999E+09,8.999999E+09,8.999999E+09,8.999999E+09,8.999999E+09]];
	LOCAL CONST Robtarget Tr_meulage_bavure_P391 :=[[218.53028125,-253.023828125,19.5],[0.749965349966833,-0.658047486126157,-0.0443684725768967,0.050565981582136],[0,0,0,0],[8.999999E+09,8.999999E+09,8.999999E+09,8.999999E+09,8.999999E+09,8.999999E+09]];
	LOCAL CONST Robtarget Tr_meulage_bavure_P392 :=[[219.095953125,-252.89653125,19.5],[0.749898043744128,-0.657704851819652,-0.0469840791912529,0.0535700306530519],[0,0,0,0],[8.999999E+09,8.999999E+09,8.999999E+09,8.999999E+09,8.999999E+09,8.999999E+09]];
	LOCAL CONST Robtarget Tr_meulage_bavure_P393 :=[[219.305234375,-252.853046875,19.5],[0.749762700654114,-0.657311062331293,-0.0501966798417859,0.0572569068114641],[0,0,0,0],[8.999999E+09,8.999999E+09,8.999999E+09,8.999999E+09,8.999999E+09,8.999999E+09]];
	LOCAL CONST Robtarget Tr_meulage_bavure_P394 :=[[219.690984375,-252.8630625,19.5],[0.749535210602135,-0.656855944291842,-0.0540977190566767,0.0617306512921282],[0,0,0,0],[8.999999E+09,8.999999E+09,8.999999E+09,8.999999E+09,8.999999E+09,8.999999E+09]];
	LOCAL CONST Robtarget Tr_meulage_bavure_P395 :=[[228.460390625,-252.180765625,19.5],[0.749188135675054,-0.656324703232434,-0.0587724428571624,0.0670881602907343],[0,0,0,0],[8.999999E+09,8.999999E+09,8.999999E+09,8.999999E+09,8.999999E+09,8.999999E+09]];
	LOCAL CONST Robtarget Tr_meulage_bavure_P396 :=[[229.2111875,-252.066453125,19.5],[0.748708072452323,-0.655680154651966,-0.0642809169024341,0.0734010951041143],[0,0,0,0],[8.999999E+09,8.999999E+09,8.999999E+09,8.999999E+09,8.999999E+09,8.999999E+09]];
	LOCAL CONST Robtarget Tr_meulage_bavure_P397 :=[[229.5289375,-252.008765625,19.5],[0.74806056809837,-0.654896048548644,-0.0706885228860066,0.0807445650425435],[0,0,0,0],[8.999999E+09,8.999999E+09,8.999999E+09,8.999999E+09,8.999999E+09,8.999999E+09]];
	LOCAL CONST Robtarget Tr_meulage_bavure_P398 :=[[230.121515625,-252.01496875,19.5],[0.747208688928678,-0.65394084858474,-0.0780370547917106,0.089167033264498],[0,0,0,0],[8.999999E+09,8.999999E+09,8.999999E+09,8.999999E+09,8.999999E+09,8.999999E+09]];
	LOCAL CONST Robtarget Tr_meulage_bavure_P399 :=[[236.2184375,-251.14521875,19.5],[0.746117745514469,-0.652768281572659,-0.0863604401454113,0.0987104593190307],[0,0,0,0],[8.999999E+09,8.999999E+09,8.999999E+09,8.999999E+09,8.999999E+09,8.999999E+09]];
	LOCAL CONST Robtarget Tr_meulage_bavure_P400 :=[[238.810796875,-250.59940625,19.5],[0.744722782324835,-0.651364765352148,-0.0956580684945637,0.109368431807295],[0,0,0,0],[8.999999E+09,8.999999E+09,8.999999E+09,8.999999E+09,8.999999E+09,8.999999E+09]];
	LOCAL CONST Robtarget Tr_meulage_bavure_P401 :=[[239.35559375,-250.46771875,19.5],[0.742983687419268,-0.649671188928834,-0.105940978225713,0.12115731772056],[0,0,0,0],[8.999999E+09,8.999999E+09,8.999999E+09,8.999999E+09,8.999999E+09,8.999999E+09]];
	LOCAL CONST Robtarget Tr_meulage_bavure_P402 :=[[239.716,-250.348359375,19.5],[0.740855170887779,-0.647644140892055,-0.117164267563178,0.134026926188045],[0,0,0,0],[8.999999E+09,8.999999E+09,8.999999E+09,8.999999E+09,8.999999E+09,8.999999E+09]];
	LOCAL CONST Robtarget Tr_meulage_bavure_P403 :=[[241.07934375,-250.016328125,19.5],[0.738280265150873,-0.64524724280864,-0.129287782215408,0.14792875010094],[0,0,0,0],[8.999999E+09,8.999999E+09,8.999999E+09,8.999999E+09,8.999999E+09,8.999999E+09]];
	LOCAL CONST Robtarget Tr_meulage_bavure_P404 :=[[242.75121875,-249.450046875,19.5],[0.735211311086142,-0.642438716951977,-0.142250856881771,0.162792864488882],[0,0,0,0],[8.999999E+09,8.999999E+09,8.999999E+09,8.999999E+09,8.999999E+09,8.999999E+09]];
	LOCAL CONST Robtarget Tr_meulage_bavure_P405 :=[[243.32434375,-249.18409375,19.5],[0.731621118403904,-0.639170970187056,-0.155958268975862,0.178516185018642],[0,0,0,0],[8.999999E+09,8.999999E+09,8.999999E+09,8.999999E+09,8.999999E+09,8.999999E+09]];
	LOCAL CONST Robtarget Tr_meulage_bavure_P406 :=[[245.67559375,-248.14575,19.5],[0.727468367521003,-0.635426308955196,-0.170310835968523,0.194980510040378],[0,0,0,0],[8.999999E+09,8.999999E+09,8.999999E+09,8.999999E+09,8.999999E+09,8.999999E+09]];
	LOCAL CONST Robtarget Tr_meulage_bavure_P407 :=[[247.46203125,-247.164203125,19.5],[0.722730926996024,-0.631180073813323,-0.185202431405251,0.212065511071603],[0,0,0,0],[8.999999E+09,8.999999E+09,8.999999E+09,8.999999E+09,8.999999E+09,8.999999E+09]];
	LOCAL CONST Robtarget Tr_meulage_bavure_P408 :=[[248.314765625,-246.66059375,19.5],[0.717389226773837,-0.626427510399991,-0.200519874230862,0.229636781812811],[0,0,0,0],[8.999999E+09,8.999999E+09,8.999999E+09,8.999999E+09,8.999999E+09,8.999999E+09]];
	LOCAL CONST Robtarget Tr_meulage_bavure_P409 :=[[249.07928125,-246.065078125,19.5],[0.711443692817404,-0.621171372251387,-0.216136121649987,0.247546309129759],[0,0,0,0],[8.999999E+09,8.999999E+09,8.999999E+09,8.999999E+09,8.999999E+09,8.999999E+09]];
	LOCAL CONST Robtarget Tr_meulage_bavure_P410 :=[[250.705390625,-244.898109375,19.5],[0.704909523264806,-0.615400954640711,-0.23194447789707,0.265680236771462],[0,0,0,0],[8.999999E+09,8.999999E+09,8.999999E+09,8.999999E+09,8.999999E+09,8.999999E+09]];
	LOCAL CONST Robtarget Tr_meulage_bavure_P411 :=[[252.961421875,-242.688328125,19.5],[0.697810666434406,-0.609150201754592,-0.247809719397606,0.283877876004435],[0,0,0,0],[8.999999E+09,8.999999E+09,8.999999E+09,8.999999E+09,8.999999E+09,8.999999E+09]];
	LOCAL CONST Robtarget Tr_meulage_bavure_P412 :=[[252.97034375,-242.6775625,19.5],[0.690175426010377,-0.602438874924228,-0.263634971066927,0.30202961004174],[0,0,0,0],[8.999999E+09,8.999999E+09,8.999999E+09,8.999999E+09,8.999999E+09,8.999999E+09]];
	LOCAL CONST Robtarget Tr_meulage_bavure_P413 :=[[252.9741875,-242.67371875,19.5],[0.68203699996809,-0.59529928452741,-0.279330073684175,0.320029689952783],[0,0,0,0],[8.999999E+09,8.999999E+09,8.999999E+09,8.999999E+09,8.999999E+09,8.999999E+09]];
	LOCAL CONST Robtarget Tr_meulage_bavure_P414 :=[[253.121828125,-242.486421875,19.5],[0.673442887212124,-0.587778927358809,-0.294798965257567,0.337763497582842],[0,0,0,0],[8.999999E+09,8.999999E+09,8.999999E+09,8.999999E+09,8.999999E+09,8.999999E+09]];
	LOCAL CONST Robtarget Tr_meulage_bavure_P415 :=[[256.936765625,-237.625578125,19.5],[0.664444277190496,-0.579915155410377,-0.309968715605778,0.355150123722154],[0,0,0,0],[8.999999E+09,8.999999E+09,8.999999E+09,8.999999E+09,8.999999E+09,8.999999E+09]];
	LOCAL CONST Robtarget Tr_meulage_bavure_P416 :=[[257.0650625,-237.44225,19.5],[0.655098546834546,-0.571760132361724,-0.324767698241302,0.372105075423618],[0,0,0,0],[8.999999E+09,8.999999E+09,8.999999E+09,8.999999E+09,8.999999E+09,8.999999E+09]];
	LOCAL CONST Robtarget Tr_meulage_bavure_P417 :=[[258.070796875,-235.771359375,19.5],[0.645473621108132,-0.563366986831293,-0.339127917112701,0.388553340529954],[0,0,0,0],[8.999999E+09,8.999999E+09,8.999999E+09,8.999999E+09,8.999999E+09,8.999999E+09]];
	LOCAL CONST Robtarget Tr_meulage_bavure_P418 :=[[258.29534375,-235.445703125,19.5],[0.63564962762985,-0.554806771591956,-0.352975995856972,0.404409376051697],[0,0,0,0],[8.999999E+09,8.999999E+09,8.999999E+09,8.999999E+09,8.999999E+09,8.999999E+09]];
	LOCAL CONST Robtarget Tr_meulage_bavure_P419 :=[[259.848578125,-232.276421875,19.5],[0.625694415013696,-0.546145633074355,-0.366268591883559,0.419617403230747],[0,0,0,0],[8.999999E+09,8.999999E+09,8.999999E+09,8.999999E+09,8.999999E+09,8.999999E+09]];
	LOCAL CONST Robtarget Tr_meulage_bavure_P420 :=[[260.437625,-230.72940625,19.5],[0.615719275836525,-0.537462316231664,-0.378924215389454,0.434097305895495],[0,0,0,0],[8.999999E+09,8.999999E+09,8.999999E+09,8.999999E+09,8.999999E+09,8.999999E+09]];
	LOCAL CONST Robtarget Tr_meulage_bavure_P421 :=[[260.9164375,-228.562140625,19.5],[0.605802260923358,-0.528849892378476,-0.390906739738155,0.447787151243432],[0,0,0,0],[8.999999E+09,8.999999E+09,8.999999E+09,8.999999E+09,8.999999E+09,8.999999E+09]];
	LOCAL CONST Robtarget Tr_meulage_bavure_P422 :=[[261.62140625,-225.82559375,19.5],[0.596053977669699,-0.520384497957173,-0.402159599448422,0.46063791264015],[0,0,0,0],[8.999999E+09,8.999999E+09,8.999999E+09,8.999999E+09,8.999999E+09,8.999999E+09]];
	LOCAL CONST Robtarget Tr_meulage_bavure_P423 :=[[261.674984375,-225.5849375,19.5],[0.586571927616722,-0.512164274610368,-0.412644872817524,0.472594264123304],[0,0,0,0],[8.999999E+09,8.999999E+09,8.999999E+09,8.999999E+09,8.999999E+09,8.999999E+09]];
	LOCAL CONST Robtarget Tr_meulage_bavure_P424 :=[[261.705875,-225.2533125,19.5],[0.577446232242933,-0.504259896560196,-0.422341115389678,0.483638075259738],[0,0,0,0],[8.999999E+09,8.999999E+09,8.999999E+09,8.999999E+09,8.999999E+09,8.999999E+09]];
	LOCAL CONST Robtarget Tr_meulage_bavure_P425 :=[[261.8955,-223.0171875,19.5],[0.568774260831843,-0.496751065917414,-0.431221215937708,0.49374333580344],[0,0,0,0],[8.999999E+09,8.999999E+09,8.999999E+09,8.999999E+09,8.999999E+09,8.999999E+09]];
	LOCAL CONST Robtarget Tr_meulage_bavure_P426 :=[[261.93596875,-222.42596875,19.5],[0.560631284286388,-0.489717190853575,-0.439281915355628,0.502892667378805],[0,0,0,0],[8.999999E+09,8.999999E+09,8.999999E+09,8.999999E+09,8.999999E+09,8.999999E+09]];
	LOCAL CONST Robtarget Tr_meulage_bavure_P427 :=[[261.94903125,-222.289375,19.5],[0.553084697490788,-0.48321826160194,-0.44652685910569,0.511088243998166],[0,0,0,0],[8.999999E+09,8.999999E+09,8.999999E+09,8.999999E+09,8.999999E+09,8.999999E+09]];
	LOCAL CONST Robtarget Tr_meulage_bavure_P428 :=[[261.718625,-218.30659375,19.5],[0.546185112110093,-0.477281663645818,-0.45297063636149,0.518364388679462],[0,0,0,0],[8.999999E+09,8.999999E+09,8.999999E+09,8.999999E+09,8.999999E+09,8.999999E+09]];
	LOCAL CONST Robtarget Tr_meulage_bavure_P429 :=[[261.438421875,-215.133671875,19.5],[0.539973468848788,-0.471950255816109,-0.45863238833589,0.524736068270358],[0,0,0,0],[8.999999E+09,8.999999E+09,8.999999E+09,8.999999E+09,8.999999E+09,8.999999E+09]];
	LOCAL CONST Robtarget Tr_meulage_bavure_P430 :=[[261.083,-211.710078125,19.5],[0.534459515930862,-0.467222237950218,-0.463551586974474,0.530260626870585],[0,0,0,0],[8.999999E+09,8.999999E+09,8.999999E+09,8.999999E+09,8.999999E+09,8.999999E+09]];
	LOCAL CONST Robtarget Tr_meulage_bavure_P431 :=[[260.944640625,-208.694359375,19.5],[0.529640022670996,-0.463107980364123,-0.467774092708536,0.534976488360784],[0,0,0,0],[8.999999E+09,8.999999E+09,8.999999E+09,8.999999E+09,8.999999E+09,8.999999E+09]];
	LOCAL CONST Robtarget Tr_meulage_bavure_P432 :=[[260.598328125,-205.40334375,19.5],[0.525494608340936,-0.45959432343791,-0.471352638878927,0.538938924452602],[0,0,0,0],[8.999999E+09,8.999999E+09,8.999999E+09,8.999999E+09,8.999999E+09,8.999999E+09]];
	LOCAL CONST Robtarget Tr_meulage_bavure_P433 :=[[260.2084375,-201.241390625,19.5],[0.521987703575286,-0.45664693800678,-0.474344411285029,0.542217475564825],[0,0,0,0],[8.999999E+09,8.999999E+09,8.999999E+09,8.999999E+09,8.999999E+09,8.999999E+09]];
	LOCAL CONST Robtarget Tr_meulage_bavure_P434 :=[[260.195921875,-200.50809375,19.5],[0.519085212413149,-0.454217346627141,-0.476795715762936,0.544888052453992],[0,0,0,0],[8.999999E+09,8.999999E+09,8.999999E+09,8.999999E+09,8.999999E+09,8.999999E+09]];
	LOCAL CONST Robtarget Tr_meulage_bavure_P435 :=[[259.918765625,-196.814125,19.5],[0.516723148049165,-0.452274054470682,-0.478779684758523,0.547005833045079],[0,0,0,0],[8.999999E+09,8.999999E+09,8.999999E+09,8.999999E+09,8.999999E+09,8.999999E+09]];
	LOCAL CONST Robtarget Tr_meulage_bavure_P436 :=[[259.669671875,-193.98465625,19.5],[0.51484572032203,-0.450758323563017,-0.480351691842957,0.548646580366959],[0,0,0,0],[8.999999E+09,8.999999E+09,8.999999E+09,8.999999E+09,8.999999E+09,8.999999E+09]];
	LOCAL CONST Robtarget Tr_meulage_bavure_P437 :=[[259.464296875,-189.94690625,19.5],[0.513380921284986,-0.449610077067721,-0.481578936167681,0.549884111881169],[0,0,0,0],[8.999999E+09,8.999999E+09,8.999999E+09,8.999999E+09,8.999999E+09,8.999999E+09]];
	LOCAL CONST Robtarget Tr_meulage_bavure_P438 :=[[258.976140625,-184.800140625,19.5],[0.512271783494415,-0.448783417508181,-0.482513610567182,0.550773709995811],[0,0,0,0],[8.999999E+09,8.999999E+09,8.999999E+09,8.999999E+09,8.999999E+09,8.999999E+09]];
	LOCAL CONST Robtarget Tr_meulage_bavure_P439 :=[[258.704828125,-181.735,19.5],[0.511460316430395,-0.448217470840244,-0.483203860536812,0.551383235792326],[0,0,0,0],[8.999999E+09,8.999999E+09,8.999999E+09,8.999999E+09,8.999999E+09,8.999999E+09]];
	LOCAL CONST Robtarget Tr_meulage_bavure_P440 :=[[258.20990625,-176.21328125,19.5],[0.510889491709968,-0.447861125841986,-0.483697423844222,0.551769101514702],[0,0,0,0],[8.999999E+09,8.999999E+09,8.999999E+09,8.999999E+09,8.999999E+09,8.999999E+09]];
	LOCAL CONST Robtarget Tr_meulage_bavure_P441 :=[[257.34125,-165.687,19.5],[0.51050825090352,-0.447677459640546,-0.484038187540179,0.551972146844416],[0,0,0,0],[8.999999E+09,8.999999E+09,8.999999E+09,8.999999E+09,8.999999E+09,8.999999E+09]];
	LOCAL CONST Robtarget Tr_meulage_bavure_P442 :=[[257.121640625,-164.09371875,19.5],[0.510273141803534,-0.447626735762147,-0.484261390001618,0.552034901377238],[0,0,0,0],[8.999999E+09,8.999999E+09,8.999999E+09,8.999999E+09,8.999999E+09,8.999999E+09]];
	LOCAL CONST Robtarget Tr_meulage_bavure_P443 :=[[257.076109375,-163.5673125,19.5],[0.51015708436177,-0.44767719358726,-0.484387379093651,0.551990712414725],[0,0,0,0],[8.999999E+09,8.999999E+09,8.999999E+09,8.999999E+09,8.999999E+09,8.999999E+09]];
	LOCAL CONST Robtarget Tr_meulage_bavure_P444 :=[[256.619453125,-157.6275,19.5],[0.510126560678324,-0.447811220191107,-0.484445741919381,0.551858973196627],[0,0,0,0],[8.999999E+09,8.999999E+09,8.999999E+09,8.999999E+09,8.999999E+09,8.999999E+09]];
	LOCAL CONST Robtarget Tr_meulage_bavure_P445 :=[[256.57703125,-157.053734375,19.5],[0.51016323520299,-0.448007825262258,-0.484450210998511,0.551661540271296],[0,0,0,0],[8.999999E+09,8.999999E+09,8.999999E+09,8.999999E+09,8.999999E+09,8.999999E+09]];
	LOCAL CONST Robtarget Tr_meulage_bavure_P446 :=[[256.189515625,-152.93125,19.5],[0.510254021356508,-0.448257026444232,-0.484411585734173,0.551409002047837],[0,0,0,0],[8.999999E+09,8.999999E+09,8.999999E+09,8.999999E+09,8.999999E+09,8.999999E+09]];
	LOCAL CONST Robtarget Tr_meulage_bavure_P447 :=[[256.1304375,-152.15665625,19.5],[0.510398913551221,-0.448553380034484,-0.484328591914577,0.551106731368268],[0,0,0,0],[8.999999E+09,8.999999E+09,8.999999E+09,8.999999E+09,8.999999E+09,8.999999E+09]];
	LOCAL CONST Robtarget Tr_meulage_bavure_P448 :=[[255.79590625,-147.699203125,19.5],[0.510589308182098,-0.448890602072979,-0.48420833394881,0.550761359460885],[0,0,0,0],[8.999999E+09,8.999999E+09,8.999999E+09,8.999999E+09,8.999999E+09,8.999999E+09]];
	LOCAL CONST Robtarget Tr_meulage_bavure_P449 :=[[255.805484375,-147.15915625,19.5],[0.510824175391296,-0.44927023760363,-0.484051982996677,0.550371323014168],[0,0,0,0],[8.999999E+09,8.999999E+09,8.999999E+09,8.999999E+09,8.999999E+09,8.999999E+09]];
	LOCAL CONST Robtarget Tr_meulage_bavure_P450 :=[[255.761171875,-146.598109375,19.5],[0.511104934598755,-0.449702595165685,-0.48386000471851,0.54992619283305],[0,0,0,0],[8.999999E+09,8.999999E+09,8.999999E+09,8.999999E+09,8.999999E+09,8.999999E+09]];
	LOCAL CONST Robtarget Tr_meulage_bavure_P451 :=[[255.310734375,-141.262296875,19.5],[0.511441208719093,-0.450188766282674,-0.483622770890847,0.549424226088272],[0,0,0,0],[8.999999E+09,8.999999E+09,8.999999E+09,8.999999E+09,8.999999E+09,8.999999E+09]];
	LOCAL CONST Robtarget Tr_meulage_bavure_P452 :=[[255.219109375,-140.926484375,19.5],[0.511837661337063,-0.450725487150289,-0.483334687495054,0.548868220554077],[0,0,0,0],[8.999999E+09,8.999999E+09,8.999999E+09,8.999999E+09,8.999999E+09,8.999999E+09]];
	LOCAL CONST Robtarget Tr_meulage_bavure_P453 :=[[254.78534375,-138.16515625,19.5],[0.512300126686561,-0.451318173730405,-0.482990681162329,0.548252212186996],[0,0,0,0],[8.999999E+09,8.999999E+09,8.999999E+09,8.999999E+09,8.999999E+09,8.999999E+09]];
	LOCAL CONST Robtarget Tr_meulage_bavure_P454 :=[[254.48925,-135.745546875,19.5],[0.512812338302095,-0.451968413003135,-0.482606831602188,0.547575296578893],[0,0,0,0],[8.999999E+09,8.999999E+09,8.999999E+09,8.999999E+09,8.999999E+09,8.999999E+09]];
	LOCAL CONST Robtarget Tr_meulage_bavure_P455 :=[[254.4350625,-134.94834375,19.5],[0.513374672713617,-0.452654958729195,-0.482178303005955,0.54685831607863],[0,0,0,0],[8.999999E+09,8.999999E+09,8.999999E+09,8.999999E+09,8.999999E+09,8.999999E+09]];
	LOCAL CONST Robtarget Tr_meulage_bavure_P456 :=[[254.3178125,-134.512328125,19.5],[0.513957946997891,-0.453365860150887,-0.481731585973282,0.546114735786379],[0,0,0,0],[8.999999E+09,8.999999E+09,8.999999E+09,8.999999E+09,8.999999E+09,8.999999E+09]];
	LOCAL CONST Robtarget Tr_meulage_bavure_P457 :=[[254.20678125,-133.525453125,19.5],[0.514533219505006,-0.454070839927623,-0.481289700052433,0.545376441530687],[0,0,0,0],[8.999999E+09,8.999999E+09,8.999999E+09,8.999999E+09,8.999999E+09,8.999999E+09]];
	LOCAL CONST Robtarget Tr_meulage_bavure_P458 :=[[253.979609375,-129.7419453125,19.5],[0.515061956640217,-0.454725073307884,-0.480882918605195,0.544690652683558],[0,0,0,0],[8.999999E+09,8.999999E+09,8.999999E+09,8.999999E+09,8.999999E+09,8.999999E+09]];
	LOCAL CONST Robtarget Tr_meulage_bavure_P459 :=[[253.770453125,-128.4891953125,19.5],[0.515494777518612,-0.455300295084152,-0.480555692825323,0.544089148706804],[0,0,0,0],[8.999999E+09,8.999999E+09,8.999999E+09,8.999999E+09,8.999999E+09,8.999999E+09]];
	LOCAL CONST Robtarget Tr_meulage_bavure_P460 :=[[253.59796875,-127.5994296875,19.5],[0.51578528300125,-0.455757319982431,-0.48034779182549,0.543614574869114],[0,0,0,0],[8.999999E+09,8.999999E+09,8.999999E+09,8.999999E+09,8.999999E+09,8.999999E+09]];
	LOCAL CONST Robtarget Tr_meulage_bavure_P461 :=[[253.554203125,-125.90103125,19.5],[0.515904008793014,-0.456058508945631,-0.480282583947883,0.543306846713651],[0,0,0,0],[8.999999E+09,8.999999E+09,8.999999E+09,8.999999E+09,8.999999E+09,8.999999E+09]];
	LOCAL CONST Robtarget Tr_meulage_bavure_P462 :=[[253.393671875,-122.855328125,19.5],[0.5158309757671,-0.456192296029593,-0.480378490996382,0.543179067040003],[0,0,0,0],[8.999999E+09,8.999999E+09,8.999999E+09,8.999999E+09,8.999999E+09,8.999999E+09]];
	LOCAL CONST Robtarget Tr_meulage_bavure_P463 :=[[253.375796875,-121.13490625,19.5],[0.515559384703303,-0.456147457257296,-0.480640604934424,0.543242696196025],[0,0,0,0],[8.999999E+09,8.999999E+09,8.999999E+09,8.999999E+09,8.999999E+09,8.999999E+09]];
	LOCAL CONST Robtarget Tr_meulage_bavure_P464 :=[[253.3749375,-118.494734375,19.5],[0.515112644458464,-0.455947333121809,-0.481049676871339,0.543472355617191],[0,0,0,0],[8.999999E+09,8.999999E+09,8.999999E+09,8.999999E+09,8.999999E+09,8.999999E+09]];
	LOCAL CONST Robtarget Tr_meulage_bavure_P465 :=[[253.4138125,-117.4678046875,19.5],[0.514520309600652,-0.455615442541134,-0.481580134764975,0.54384188265179],[0,0,0,0],[8.999999E+09,8.999999E+09,8.999999E+09,8.999999E+09,8.999999E+09,8.999999E+09]];
	LOCAL CONST Robtarget Tr_meulage_bavure_P466 :=[[253.27503125,-115.280546875,19.5],[0.513822616760244,-0.455187278871185,-0.482197809379712,0.544312531813211],[0,0,0,0],[8.999999E+09,8.999999E+09,8.999999E+09,8.999999E+09,8.999999E+09,8.999999E+09]];
	LOCAL CONST Robtarget Tr_meulage_bavure_P467 :=[[253.19903125,-114.1990546875,19.5],[0.513057661643815,-0.454700937075843,-0.482871224194724,0.544843348583443],[0,0,0,0],[8.999999E+09,8.999999E+09,8.999999E+09,8.999999E+09,8.999999E+09,8.999999E+09]];
	LOCAL CONST Robtarget Tr_meulage_bavure_P468 :=[[253.053046875,-113.1082734375,19.5],[0.512271684274364,-0.454195425499588,-0.483561194356519,0.545392343417518],[0,0,0,0],[8.999999E+09,8.999999E+09,8.999999E+09,8.999999E+09,8.999999E+09,8.999999E+09]];
	LOCAL CONST Robtarget Tr_meulage_bavure_P469 :=[[252.494453125,-109.2521484375,19.5],[0.511491825814146,-0.45370132911826,-0.484246264330221,0.545927441665887],[0,0,0,0],[8.999999E+09,8.999999E+09,8.999999E+09,8.999999E+09,8.999999E+09,8.999999E+09]];
	LOCAL CONST Robtarget Tr_meulage_bavure_P470 :=[[251.9350625,-104.8428515625,19.5],[0.510764530279985,-0.453236348302999,-0.484883594578379,0.546428684178986],[0,0,0,0],[8.999999E+09,8.999999E+09,8.999999E+09,8.999999E+09,8.999999E+09,8.999999E+09]];
	LOCAL CONST Robtarget Tr_meulage_bavure_P471 :=[[251.55846875,-100.7880078125,19.5],[0.510102495405296,-0.452836271462604,-0.485467438572106,0.546860239472003],[0,0,0,0],[8.999999E+09,8.999999E+09,8.999999E+09,8.999999E+09,8.999999E+09,8.999999E+09]];
	LOCAL CONST Robtarget Tr_meulage_bavure_P472 :=[[251.184390625,-96.444609375,19.5],[0.509532235996624,-0.452506423741794,-0.485972708180077,0.547216012061795],[0,0,0,0],[8.999999E+09,8.999999E+09,8.999999E+09,8.999999E+09,8.999999E+09,8.999999E+09]];
	LOCAL CONST Robtarget Tr_meulage_bavure_P473 :=[[250.968875,-90.9879921875,19.5],[0.509061772506297,-0.452269380046939,-0.486395978513014,0.547473717845042],[0,0,0,0],[8.999999E+09,8.999999E+09,8.999999E+09,8.999999E+09,8.999999E+09,8.999999E+09]];
	LOCAL CONST Robtarget Tr_meulage_bavure_P474 :=[[250.867671875,-89.68565625,19.5],[0.508691365717335,-0.452131132212908,-0.486738377012331,0.54762787189104],[0,0,0,0],[8.999999E+09,8.999999E+09,8.999999E+09,8.999999E+09,8.999999E+09,8.999999E+09]];
	LOCAL CONST Robtarget Tr_meulage_bavure_P475 :=[[250.543390625,-87.3466015625,19.5],[0.508435177343764,-0.452086734603547,-0.486984994698522,0.547683183759916],[0,0,0,0],[8.999999E+09,8.999999E+09,8.999999E+09,8.999999E+09,8.999999E+09,8.999999E+09]];
	LOCAL CONST Robtarget Tr_meulage_bavure_P476 :=[[249.9633125,-84.026,19.5],[0.508286613160854,-0.452132436782303,-0.487141708823111,0.547643984734302],[0,0,0,0],[8.999999E+09,8.999999E+09,8.999999E+09,8.999999E+09,8.999999E+09,8.999999E+09]];
	LOCAL CONST Robtarget Tr_meulage_bavure_P477 :=[[249.2368125,-80.2268671875,19.5],[0.508245757705925,-0.452269251091675,-0.487208563652574,0.547509442653277],[0,0,0,0],[8.999999E+09,8.999999E+09,8.999999E+09,8.999999E+09,8.999999E+09,8.999999E+09]];
	LOCAL CONST Robtarget Tr_meulage_bavure_P478 :=[[249.060734375,-78.9468828125,19.5],[0.508298900835706,-0.452483212842013,-0.487196400410689,0.547294104602132],[0,0,0,0],[8.999999E+09,8.999999E+09,8.999999E+09,8.999999E+09,8.999999E+09,8.999999E+09]];
	LOCAL CONST Robtarget Tr_meulage_bavure_P479 :=[[248.887515625,-76.2736796875,19.5],[0.508428315933993,-0.452768661042142,-0.487121602255483,0.547004325166338],[0,0,0,0],[8.999999E+09,8.999999E+09,8.999999E+09,8.999999E+09,8.999999E+09,8.999999E+09]];
	LOCAL CONST Robtarget Tr_meulage_bavure_P480 :=[[248.61584375,-73.7588984375,19.5],[0.508627179667676,-0.453111766779385,-0.486988125238063,0.546654081468789],[0,0,0,0],[8.999999E+09,8.999999E+09,8.999999E+09,8.999999E+09,8.999999E+09,8.999999E+09]];
	LOCAL CONST Robtarget Tr_meulage_bavure_P481 :=[[248.5808125,-71.612640625,19.5],[0.508876115523772,-0.453493900093349,-0.48681156612789,0.546262648102239],[0,0,0,0],[8.999999E+09,8.999999E+09,8.999999E+09,8.999999E+09,8.999999E+09,8.999999E+09]];
	LOCAL CONST Robtarget Tr_meulage_bavure_P482 :=[[248.230046875,-68.2864375,19.5],[0.509170168081714,-0.453906942843495,-0.486595186887367,0.545838209794954],[0,0,0,0],[8.999999E+09,8.999999E+09,8.999999E+09,8.999999E+09,8.999999E+09,8.999999E+09]];
	LOCAL CONST Robtarget Tr_meulage_bavure_P483 :=[[248.0520625,-66.376859375,19.5],[0.509481151615789,-0.454341273629273,-0.486365148466733,0.545391515869207],[0,0,0,0],[8.999999E+09,8.999999E+09,8.999999E+09,8.999999E+09,8.999999E+09,8.999999E+09]];
	LOCAL CONST Robtarget Tr_meulage_bavure_P484 :=[[247.206546875,-55.03701953125,19.5],[0.509810675751206,-0.454778449357137,-0.486116404996158,0.544940801999655],[0,0,0,0],[8.999999E+09,8.999999E+09,8.999999E+09,8.999999E+09,8.999999E+09,8.999999E+09]];
	LOCAL CONST Robtarget Tr_meulage_bavure_P485 :=[[247.11340625,-52.98913671875,19.5],[0.510130026661102,-0.455217410851161,-0.485877343615665,0.544488449572343],[0,0,0,0],[8.999999E+09,8.999999E+09,8.999999E+09,8.999999E+09,8.999999E+09,8.999999E+09]];
	LOCAL CONST Robtarget Tr_meulage_bavure_P486 :=[[246.89434375,-50.01998828125,19.5],[0.510442670843544,-0.455647948232384,-0.485642693110643,0.544044485021188],[0,0,0,0],[8.999999E+09,8.999999E+09,8.999999E+09,8.999999E+09,8.999999E+09,8.999999E+09]];
	LOCAL CONST Robtarget Tr_meulage_bavure_P487 :=[[246.44775,-44.65310546875,19.5],[0.510734142034772,-0.45604796717706,-0.485423023077471,0.543631655130572],[0,0,0,0],[8.999999E+09,8.999999E+09,8.999999E+09,8.999999E+09,8.999999E+09,8.999999E+09]];
	LOCAL CONST Robtarget Tr_meulage_bavure_P488 :=[[246.313109375,-41.28994921875,19.5],[0.510998316354166,-0.456421950061962,-0.48522535660907,0.543245872039949],[0,0,0,0],[8.999999E+09,8.999999E+09,8.999999E+09,8.999999E+09,8.999999E+09,8.999999E+09]];
	LOCAL CONST Robtarget Tr_meulage_bavure_P489 :=[[246.02965625,-36.7373359375,19.5],[0.511230466024334,-0.456762017434207,-0.48505315722834,0.542895298101571],[0,0,0,0],[8.999999E+09,8.999999E+09,8.999999E+09,8.999999E+09,8.999999E+09,8.999999E+09]];
	LOCAL CONST Robtarget Tr_meulage_bavure_P490 :=[[245.42346875,-29.136109375,19.5],[0.511423843175751,-0.457060608671957,-0.484911985801616,0.54258789026083],[0,0,0,0],[8.999999E+09,8.999999E+09,8.999999E+09,8.999999E+09,8.999999E+09,8.999999E+09]];
	LOCAL CONST Robtarget Tr_meulage_bavure_P491 :=[[245.404609375,-28.95300390625,19.5],[0.511584839348576,-0.457322070553497,-0.484796369229515,0.542319053985044],[0,0,0,0],[8.999999E+09,8.999999E+09,8.999999E+09,8.999999E+09,8.999999E+09,8.999999E+09]];
	LOCAL CONST Robtarget Tr_meulage_bavure_P492 :=[[245.3931875,-28.7763359375,19.5],[0.511699359145338,-0.45755267624031,-0.484721517920652,0.542083355564695],[0,0,0,0],[8.999999E+09,8.999999E+09,8.999999E+09,8.999999E+09,8.999999E+09,8.999999E+09]];
	LOCAL CONST Robtarget Tr_meulage_bavure_P493 :=[[245.344484375,-28.214080078125,19.5],[0.511789186462596,-0.457739191359912,-0.484663603703605,0.541892842320474],[0,0,0,0],[8.999999E+09,8.999999E+09,8.999999E+09,8.999999E+09,8.999999E+09,8.999999E+09]];
	LOCAL CONST Robtarget Tr_meulage_bavure_P494 :=[[245.38678125,-28.603943359375,19.5],[0.511847528425695,-0.457900696612118,-0.484632692375863,0.541728911142064],[0,0,0,0],[8.999999E+09,8.999999E+09,8.999999E+09,8.999999E+09,8.999999E+09,8.999999E+09]];
	LOCAL CONST Robtarget Tr_meulage_bavure_P495 :=[[245.03009375,-22.7691953125,19.5],[0.511885743394977,-0.458042631351514,-0.484618436889807,0.541585546520615],[0,0,0,0],[8.999999E+09,8.999999E+09,8.999999E+09,8.999999E+09,8.999999E+09,8.999999E+09]];
	LOCAL CONST Robtarget Tr_meulage_bavure_P496 :=[[244.9035,-21.606720703125,19.5],[0.511919184260064,-0.458167604330563,-0.484606023558109,0.541459321703579],[0,0,0,0],[8.999999E+09,8.999999E+09,8.999999E+09,8.999999E+09,8.999999E+09,8.999999E+09]];
	LOCAL CONST Robtarget Tr_meulage_bavure_P497 :=[[244.147578125,-17.4111015625,19.5],[0.511947733841283,-0.458297334998996,-0.484599206865932,0.54132862408384],[0,0,0,0],[8.999999E+09,8.999999E+09,8.999999E+09,8.999999E+09,8.999999E+09,8.999999E+09]];
	LOCAL CONST Robtarget Tr_meulage_bavure_P498 :=[[243.853828125,-15.1081240234375,19.5],[0.511989407036485,-0.45842788240118,-0.484579393258657,0.541196392586528],[0,0,0,0],[8.999999E+09,8.999999E+09,8.999999E+09,8.999999E+09,8.999999E+09,8.999999E+09]];
	LOCAL CONST Robtarget Tr_meulage_bavure_P499 :=[[243.707828125,-13.1136171875,19.5],[0.512048482453559,-0.458563486194833,-0.484543022440916,0.541058167066787],[0,0,0,0],[8.999999E+09,8.999999E+09,8.999999E+09,8.999999E+09,8.999999E+09,8.999999E+09]];
	LOCAL CONST Robtarget Tr_meulage_bavure_P500 :=[[243.479375,-9.506896484375,19.5],[0.512121497307507,-0.458717022831825,-0.484495652269734,0.540901310676494],[0,0,0,0],[8.999999E+09,8.999999E+09,8.999999E+09,8.999999E+09,8.999999E+09,8.999999E+09]];
	LOCAL CONST Robtarget Tr_meulage_bavure_P501 :=[[243.0883125,-4.215484375,19.5],[0.512212345697298,-0.458877639185891,-0.48443159426934,0.540736401256768],[0,0,0,0],[8.999999E+09,8.999999E+09,8.999999E+09,8.999999E+09,8.999999E+09,8.999999E+09]];
	LOCAL CONST Robtarget Tr_meulage_bavure_P502 :=[[242.870546875,-1.85137939453125,19.5],[0.512324221585642,-0.459043109611235,-0.484347292239219,0.540565459491864],[0,0,0,0],[8.999999E+09,8.999999E+09,8.999999E+09,8.999999E+09,8.999999E+09,8.999999E+09]];
	LOCAL CONST Robtarget Tr_meulage_bavure_P503 :=[[242.6455625,0.43963623046875,19.5],[0.512437921588957,-0.459209835152059,-0.484261267531771,0.540393124110338],[0,0,0,0],[8.999999E+09,8.999999E+09,8.999999E+09,8.999999E+09,8.999999E+09,8.999999E+09]];
	LOCAL CONST Robtarget Tr_meulage_bavure_P504 :=[[242.52465625,2.1629638671875,19.5],[0.512549890338318,-0.459377517981263,-0.484177008447211,0.540219890765475],[0,0,0,0],[8.999999E+09,8.999999E+09,8.999999E+09,8.999999E+09,8.999999E+09,8.999999E+09]];
	LOCAL CONST Robtarget Tr_meulage_bavure_P505 :=[[242.3305625,6.36117578125,19.5],[0.512649217181834,-0.459516766454861,-0.484100635058017,0.540075639708131],[0,0,0,0],[8.999999E+09,8.999999E+09,8.999999E+09,8.999999E+09,8.999999E+09,8.999999E+09]];
	LOCAL CONST Robtarget Tr_meulage_bavure_P506 :=[[242.28234375,10.177185546875,19.5],[0.512722015426519,-0.459630451173285,-0.48404647991849,0.539958321104259],[0,0,0,0],[8.999999E+09,8.999999E+09,8.999999E+09,8.999999E+09,8.999999E+09,8.999999E+09]];
	LOCAL CONST Robtarget Tr_meulage_bavure_P507 :=[[242.124578125,15.8605654296875,19.5],[0.512754120796776,-0.459700699366845,-0.484025808854329,0.539886557501177],[0,0,0,0],[8.999999E+09,8.999999E+09,8.999999E+09,8.999999E+09,8.999999E+09,8.999999E+09]];
	LOCAL CONST Robtarget Tr_meulage_bavure_P508 :=[[242.06921875,18.71090625,19.5],[0.512732227437486,-0.45972066141866,-0.484050804833027,0.539867941956441],[0,0,0,0],[8.999999E+09,8.999999E+09,8.999999E+09,8.999999E+09,8.999999E+09,8.999999E+09]];
	LOCAL CONST Robtarget Tr_meulage_bavure_P509 :=[[241.778203125,22.2959296875,19.5],[0.512645581937505,-0.459679030880278,-0.484130369384253,0.539914327767649],[0,0,0,0],[8.999999E+09,8.999999E+09,8.999999E+09,8.999999E+09,8.999999E+09,8.999999E+09]];
	LOCAL CONST Robtarget Tr_meulage_bavure_P510 :=[[241.72503125,23.72668359375,19.5],[0.512490373763828,-0.459569372300866,-0.484267230279388,0.540032275442802],[0,0,0,0],[8.999999E+09,8.999999E+09,8.999999E+09,8.999999E+09,8.999999E+09,8.999999E+09]];
	LOCAL CONST Robtarget Tr_meulage_bavure_P511 :=[[241.673515625,25.2835703125,19.5],[0.512251657083112,-0.459380051283766,-0.48447429597248,0.540234083375068],[0,0,0,0],[8.999999E+09,8.999999E+09,8.999999E+09,8.999999E+09,8.999999E+09,8.999999E+09]];
	LOCAL CONST Robtarget Tr_meulage_bavure_P512 :=[[241.49346875,28.662810546875,19.5],[0.511928395887919,-0.459112927589211,-0.484752724429148,0.540517745650043],[0,0,0,0],[8.999999E+09,8.999999E+09,8.999999E+09,8.999999E+09,8.999999E+09,8.999999E+09]];
	LOCAL CONST Robtarget Tr_meulage_bavure_P513 :=[[241.405328125,31.87676953125,19.5],[0.511527535791102,-0.458764806924322,-0.485094832233329,0.540885788125082],[0,0,0,0],[8.999999E+09,8.999999E+09,8.999999E+09,8.999999E+09,8.999999E+09,8.999999E+09]];
	LOCAL CONST Robtarget Tr_meulage_bavure_P514 :=[[241.317078125,33.58596875,19.5],[0.511041170392421,-0.458331253308941,-0.485507422747279,0.541342707405849],[0,0,0,0],[8.999999E+09,8.999999E+09,8.999999E+09,8.999999E+09,8.999999E+09,8.999999E+09]];
	LOCAL CONST Robtarget Tr_meulage_bavure_P515 :=[[241.1148125,36.7861640625,19.5],[0.510478753963318,-0.457836228659856,-0.485984680510327,0.541863746515536],[0,0,0,0],[8.999999E+09,8.999999E+09,8.999999E+09,8.999999E+09,8.999999E+09,8.999999E+09]];
	LOCAL CONST Robtarget Tr_meulage_bavure_P516 :=[[240.89478125,40.4691171875,19.5],[0.509864525664394,-0.457283621364188,-0.486502777395659,0.542443455751276],[0,0,0,0],[8.999999E+09,8.999999E+09,8.999999E+09,8.999999E+09,8.999999E+09,8.999999E+09]];
	LOCAL CONST Robtarget Tr_meulage_bavure_P517 :=[[240.710578125,42.8906875,19.5],[0.509187659305522,-0.456669871291295,-0.48707151016792,0.543085536769758],[0,0,0,0],[8.999999E+09,8.999999E+09,8.999999E+09,8.999999E+09,8.999999E+09,8.999999E+09]];
	LOCAL CONST Robtarget Tr_meulage_bavure_P518 :=[[240.57140625,43.3461015625,19.5],[0.508482791679219,-0.456028614624285,-0.487661851642402,0.543754606107081],[0,0,0,0],[8.999999E+09,8.999999E+09,8.999999E+09,8.999999E+09,8.999999E+09,8.999999E+09]];
	LOCAL CONST Robtarget Tr_meulage_bavure_P519 :=[[240.422421875,45.16003515625,19.5],[0.50776257308916,-0.455360439004472,-0.488261100802514,0.544449389202199],[0,0,0,0],[8.999999E+09,8.999999E+09,8.999999E+09,8.999999E+09,8.999999E+09,8.999999E+09]];
	LOCAL CONST Robtarget Tr_meulage_bavure_P520 :=[[240.17078125,53.7380390625,19.5],[0.507047981470274,-0.454692295202097,-0.488853028382991,0.545142162936925],[0,0,0,0],[8.999999E+09,8.999999E+09,8.999999E+09,8.999999E+09,8.999999E+09,8.999999E+09]];
	LOCAL CONST Robtarget Tr_meulage_bavure_P521 :=[[240.125671875,54.63973828125,19.5],[0.506347618131465,-0.454038501796344,-0.489431698661347,0.545818413801323],[0,0,0,0],[8.999999E+09,8.999999E+09,8.999999E+09,8.999999E+09,8.999999E+09,8.999999E+09]];
	LOCAL CONST Robtarget Tr_meulage_bavure_P522 :=[[239.96753125,56.70309375,19.5],[0.505713086840009,-0.453441908179971,-0.48995376925675,0.546433906063633],[0,0,0,0],[8.999999E+09,8.999999E+09,8.999999E+09,8.999999E+09,8.999999E+09,8.999999E+09]];
	LOCAL CONST Robtarget Tr_meulage_bavure_P523 :=[[239.359734375,60.3229375,19.5],[0.505163286934352,-0.45291856358014,-0.490403815404447,0.5469725094874],[0,0,0,0],[8.999999E+09,8.999999E+09,8.999999E+09,8.999999E+09,8.999999E+09,8.999999E+09]];
	LOCAL CONST Robtarget Tr_meulage_bavure_P524 :=[[239.26146875,61.2630625,19.5],[0.504734318664852,-0.452499633693838,-0.49075220798583,0.547402611818671],[0,0,0,0],[8.999999E+09,8.999999E+09,8.999999E+09,8.999999E+09,8.999999E+09,8.999999E+09]];
	LOCAL CONST Robtarget Tr_meulage_bavure_P525 :=[[239.1820625,61.84655859375,19.5],[0.504481103146449,-0.452225743812961,-0.490952451601655,0.547682739793103],[0,0,0,0],[8.999999E+09,8.999999E+09,8.999999E+09,8.999999E+09,8.999999E+09,8.999999E+09]];
	LOCAL CONST Robtarget Tr_meulage_bavure_P526 :=[[237.60828125,68.8543984375,19.5],[0.504414536573453,-0.452109728367448,-0.490996596897797,0.547800247027767],[0,0,0,0],[8.999999E+09,8.999999E+09,8.999999E+09,8.999999E+09,8.999999E+09,8.999999E+09]];
	LOCAL CONST Robtarget Tr_meulage_bavure_P527 :=[[237.53271875,70.44546875,19.5],[0.504591398378384,-0.452212547760151,-0.490839916716845,0.547692896145478],[0,0,0,0],[8.999999E+09,8.999999E+09,8.999999E+09,8.999999E+09,8.999999E+09,8.999999E+09]];
	LOCAL CONST Robtarget Tr_meulage_bavure_P528 :=[[237.3570625,75.94525,19.5],[0.505041505718573,-0.452560438352761,-0.490457425510222,0.547333208293959],[0,0,0,0],[8.999999E+09,8.999999E+09,8.999999E+09,8.999999E+09,8.999999E+09,8.999999E+09]];
	LOCAL CONST Robtarget Tr_meulage_bavure_P529 :=[[237.123109375,78.8272734375,19.5],[0.505758800194462,-0.453144013089005,-0.489852450097518,0.546729472921397],[0,0,0,0],[8.999999E+09,8.999999E+09,8.999999E+09,8.999999E+09,8.999999E+09,8.999999E+09]];
	LOCAL CONST Robtarget Tr_meulage_bavure_P530 :=[[236.91815625,80.8139921875,19.5],[0.50678016138542,-0.453994609085038,-0.488992456101265,0.54584717716953],[0,0,0,0],[8.999999E+09,8.999999E+09,8.999999E+09,8.999999E+09,8.999999E+09,8.999999E+09]];
	LOCAL CONST Robtarget Tr_meulage_bavure_P531 :=[[236.624203125,85.0335078125,19.5],[0.50808785659087,-0.455092197464047,-0.487888932123214,0.544703783449234],[0,0,0,0],[8.999999E+09,8.999999E+09,8.999999E+09,8.999999E+09,8.999999E+09,8.999999E+09]];
	LOCAL CONST Robtarget Tr_meulage_bavure_P532 :=[[236.409796875,88.8693515625,19.5],[0.50964010907195,-0.456409155478337,-0.486575563774014,0.543324822512908],[0,0,0,0],[8.999999E+09,8.999999E+09,8.999999E+09,8.999999E+09,8.999999E+09,8.999999E+09]];
	LOCAL CONST Robtarget Tr_meulage_bavure_P533 :=[[236.193421875,91.4233125,19.5],[0.511390106587433,-0.457899832639596,-0.485087913373024,0.541754204831424],[0,0,0,0],[8.999999E+09,8.999999E+09,8.999999E+09,8.999999E+09,8.999999E+09,8.999999E+09]];
	LOCAL CONST Robtarget Tr_meulage_bavure_P534 :=[[235.963625,95.399234375,19.5],[0.513295241180999,-0.459525725808753,-0.483459096854568,0.540029077336994],[0,0,0,0],[8.999999E+09,8.999999E+09,8.999999E+09,8.999999E+09,8.999999E+09,8.999999E+09]];
	LOCAL CONST Robtarget Tr_meulage_bavure_P535 :=[[235.47259375,100.6566484375,19.5],[0.515240968723578,-0.461188785678783,-0.481785285177944,0.538251416253526],[0,0,0,0],[8.999999E+09,8.999999E+09,8.999999E+09,8.999999E+09,8.999999E+09,8.999999E+09]];
	LOCAL CONST Robtarget Tr_meulage_bavure_P536 :=[[235.26140625,103.021515625,19.5],[0.517190105880869,-0.462846313577147,-0.480096321902974,0.536465475200611],[0,0,0,0],[8.999999E+09,8.999999E+09,8.999999E+09,8.999999E+09,8.999999E+09,8.999999E+09]];
	LOCAL CONST Robtarget Tr_meulage_bavure_P537 :=[[234.6015,104.932125,19.5],[0.519016396764805,-0.464389496060884,-0.478502446520844,0.534789476814161],[0,0,0,0],[8.999999E+09,8.999999E+09,8.999999E+09,8.999999E+09,8.999999E+09,8.999999E+09]];
	LOCAL CONST Robtarget Tr_meulage_bavure_P538 :=[[234.867671875,108.548890625,19.5],[0.520637328932792,-0.465740650787515,-0.477077240313123,0.533310158070296],[0,0,0,0],[8.999999E+09,8.999999E+09,8.999999E+09,8.999999E+09,8.999999E+09,8.999999E+09]];
	LOCAL CONST Robtarget Tr_meulage_bavure_P539 :=[[234.843140625,108.7029453125,19.5],[0.52197125989465,-0.466830880026136,-0.475895973963196,0.532107090033234],[0,0,0,0],[8.999999E+09,8.999999E+09,8.999999E+09,8.999999E+09,8.999999E+09,8.999999E+09]];
	LOCAL CONST Robtarget Tr_meulage_bavure_P540 :=[[234.786015625,109.15115625,19.5],[0.522951117869964,-0.467609967165363,-0.475022387927412,0.531240790879148],[0,0,0,0],[8.999999E+09,8.999999E+09,8.999999E+09,8.999999E+09,8.999999E+09,8.999999E+09]];
	LOCAL CONST Robtarget Tr_meulage_bavure_P541 :=[[232.831171875,117.856203125,19.5],[0.523532538976908,-0.468021310762285,-0.474496462094559,0.530775697224818],[0,0,0,0],[8.999999E+09,8.999999E+09,8.999999E+09,8.999999E+09,8.999999E+09,8.999999E+09]];
	LOCAL CONST Robtarget Tr_meulage_bavure_P542 :=[[232.7579375,120.820859375,19.5],[0.523679664619518,-0.468045192978537,-0.474353236840977,0.530737517886348],[0,0,0,0],[8.999999E+09,8.999999E+09,8.999999E+09,8.999999E+09,8.999999E+09,8.999999E+09]];
	LOCAL CONST Robtarget Tr_meulage_bavure_P543 :=[[232.63,122.4965234375,19.5],[0.523386562633535,-0.467668426845138,-0.474597042545023,0.531140655377052],[0,0,0,0],[8.999999E+09,8.999999E+09,8.999999E+09,8.999999E+09,8.999999E+09,8.999999E+09]];
	LOCAL CONST Robtarget Tr_meulage_bavure_P544 :=[[232.359015625,125.9118359375,19.5],[0.522677947477149,-0.466918074783706,-0.475204946617665,0.531954446707098],[0,0,0,0],[8.999999E+09,8.999999E+09,8.999999E+09,8.999999E+09,8.999999E+09,8.999999E+09]];
	LOCAL CONST Robtarget Tr_meulage_bavure_P545 :=[[232.17084375,127.503359375,19.5],[0.521581004592166,-0.465829384551997,-0.476151189090682,0.533138148385636],[0,0,0,0],[8.999999E+09,8.999999E+09,8.999999E+09,8.999999E+09,8.999999E+09,8.999999E+09]];
	LOCAL CONST Robtarget Tr_meulage_bavure_P546 :=[[231.954890625,130.9570625,19.5],[0.520171807686431,-0.464463605667571,-0.477364215886499,0.534619729237126],[0,0,0,0],[8.999999E+09,8.999999E+09,8.999999E+09,8.999999E+09,8.999999E+09,8.999999E+09]];
	LOCAL CONST Robtarget Tr_meulage_bavure_P547 :=[[231.87,132.390375,19.5],[0.518528888298165,-0.462880851331599,-0.478770188674934,0.536328458975441],[0,0,0,0],[8.999999E+09,8.999999E+09,8.999999E+09,8.999999E+09,8.999999E+09,8.999999E+09]];
	LOCAL CONST Robtarget Tr_meulage_bavure_P548 :=[[231.280515625,138.66815625,19.5],[0.516749018753205,-0.461172677074415,-0.480282882182785,0.538162212181248],[0,0,0,0],[8.999999E+09,8.999999E+09,8.999999E+09,8.999999E+09,8.999999E+09,8.999999E+09]];
	LOCAL CONST Robtarget Tr_meulage_bavure_P549 :=[[231.02740625,142.039609375,19.5],[0.514906695421224,-0.459398050419409,-0.481835230211509,0.54005493906478],[0,0,0,0],[8.999999E+09,8.999999E+09,8.999999E+09,8.999999E+09,8.999999E+09,8.999999E+09]];
	LOCAL CONST Robtarget Tr_meulage_bavure_P550 :=[[230.7731875,144.143953125,19.5],[0.513059660935821,-0.457632306233649,-0.483381191502051,0.541927190971029],[0,0,0,0],[8.999999E+09,8.999999E+09,8.999999E+09,8.999999E+09,8.999999E+09,8.999999E+09]];
	LOCAL CONST Robtarget Tr_meulage_bavure_P551 :=[[230.673515625,145.508703125,19.5],[0.51127044591823,-0.45592636072404,-0.484867794455649,0.543725028509099],[0,0,0,0],[8.999999E+09,8.999999E+09,8.999999E+09,8.999999E+09,8.999999E+09,8.999999E+09]];
	LOCAL CONST Robtarget Tr_meulage_bavure_P552 :=[[230.237421875,148.758546875,19.5],[0.509620690204448,-0.454339376876574,-0.486225856057069,0.545386926536123],[0,0,0,0],[8.999999E+09,8.999999E+09,8.999999E+09,8.999999E+09,8.999999E+09,8.999999E+09]];
	LOCAL CONST Robtarget Tr_meulage_bavure_P553 :=[[229.349484375,154.043578125,19.5],[0.508094493975102,-0.452853922076508,-0.487470198362082,0.546933374517356],[0,0,0,0],[8.999999E+09,8.999999E+09,8.999999E+09,8.999999E+09,8.999999E+09,8.999999E+09]];
	LOCAL CONST Robtarget Tr_meulage_bavure_P554 :=[[229.24340625,155.281734375,19.5],[0.506738103384784,-0.451526446138598,-0.488567499331369,0.54830845480672],[0,0,0,0],[8.999999E+09,8.999999E+09,8.999999E+09,8.999999E+09,8.999999E+09,8.999999E+09]];
	LOCAL CONST Robtarget Tr_meulage_bavure_P555 :=[[229.07421875,157.357328125,19.5],[0.505531098917366,-0.450332211010535,-0.489535654439026,0.549539853683714],[0,0,0,0],[8.999999E+09,8.999999E+09,8.999999E+09,8.999999E+09,8.999999E+09,8.999999E+09]];
	LOCAL CONST Robtarget Tr_meulage_bavure_P556 :=[[228.27184375,164.70971875,19.5],[0.504465594023082,-0.449255779436954,-0.490381238231134,0.550645031104735],[0,0,0,0],[8.999999E+09,8.999999E+09,8.999999E+09,8.999999E+09,8.999999E+09,8.999999E+09]];
	LOCAL CONST Robtarget Tr_meulage_bavure_P557 :=[[228.2241875,165.464140625,19.5],[0.503525304490269,-0.44830536961144,-0.491123657108887,0.551617727002609],[0,0,0,0],[8.999999E+09,8.999999E+09,8.999999E+09,8.999999E+09,8.999999E+09,8.999999E+09]];
	LOCAL CONST Robtarget Tr_meulage_bavure_P558 :=[[228.1720625,166.332734375,19.5],[0.5026999864384,-0.447452687757191,-0.491768552592605,0.552487562334821],[0,0,0,0],[8.999999E+09,8.999999E+09,8.999999E+09,8.999999E+09,8.999999E+09,8.999999E+09]];
	LOCAL CONST Robtarget Tr_meulage_bavure_P559 :=[[227.663703125,171.817171875,19.5],[0.501943079216339,-0.446664212621073,-0.492356160113411,0.553289831814027],[0,0,0,0],[8.999999E+09,8.999999E+09,8.999999E+09,8.999999E+09,8.999999E+09,8.999999E+09]];
	LOCAL CONST Robtarget Tr_meulage_bavure_P560 :=[[227.562921875,172.921171875,19.5],[0.50126471125819,-0.445949317901982,-0.492878988456167,0.554015521306422],[0,0,0,0],[8.999999E+09,8.999999E+09,8.999999E+09,8.999999E+09,8.999999E+09,8.999999E+09]];
	LOCAL CONST Robtarget Tr_meulage_bavure_P561 :=[[227.0751875,175.849453125,19.5],[0.500649976981145,-0.445290123616966,-0.493348589550587,0.554683220898571],[0,0,0,0],[8.999999E+09,8.999999E+09,8.999999E+09,8.999999E+09,8.999999E+09,8.999999E+09]];
	LOCAL CONST Robtarget Tr_meulage_bavure_P562 :=[[227.11053125,176.77584375,19.5],[0.500067315681953,-0.444656103793948,-0.493790105549809,0.555324194328448],[0,0,0,0],[8.999999E+09,8.999999E+09,8.999999E+09,8.999999E+09,8.999999E+09,8.999999E+09]];
	LOCAL CONST Robtarget Tr_meulage_bavure_P563 :=[[226.5859375,183.604125,19.5],[0.499532558378882,-0.444063625046591,-0.49419158791415,0.555922111868938],[0,0,0,0],[8.999999E+09,8.999999E+09,8.999999E+09,8.999999E+09,8.999999E+09,8.999999E+09]];
	LOCAL CONST Robtarget Tr_meulage_bavure_P564 :=[[226.35021875,185.873875,19.5],[0.499020302881344,-0.443497007461827,-0.494575127966217,0.556493112699355],[0,0,0,0],[8.999999E+09,8.999999E+09,8.999999E+09,8.999999E+09,8.999999E+09,8.999999E+09]];
	LOCAL CONST Robtarget Tr_meulage_bavure_P565 :=[[226.078859375,192.22165625,19.5],[0.498533405937362,-0.442953161133395,-0.494937332481511,0.557040372973551],[0,0,0,0],[8.999999E+09,8.999999E+09,8.999999E+09,8.999999E+09,8.999999E+09,8.999999E+09]];
	LOCAL CONST Robtarget Tr_meulage_bavure_P566 :=[[226.0784375,192.23453125,19.5],[0.498074226080976,-0.442438946608891,-0.495277575103297,0.557557142755117],[0,0,0,0],[8.999999E+09,8.999999E+09,8.999999E+09,8.999999E+09,8.999999E+09,8.999999E+09]];
	LOCAL CONST Robtarget Tr_meulage_bavure_P567 :=[[226.07659375,192.252875,19.5],[0.497618065995628,-0.441918777829087,-0.49561239759693,0.558079210816027],[0,0,0,0],[8.999999E+09,8.999999E+09,8.999999E+09,8.999999E+09,8.999999E+09,8.999999E+09]];
	LOCAL CONST Robtarget Tr_meulage_bavure_P568 :=[[226.068046875,192.3241875,19.5],[0.497161904177804,-0.441396725817617,-0.495945742743777,0.558602534657792],[0,0,0,0],[8.999999E+09,8.999999E+09,8.999999E+09,8.999999E+09,8.999999E+09,8.999999E+09]];
	LOCAL CONST Robtarget Tr_meulage_bavure_P569 :=[[225.591375,195.7669375,19.5],[0.496660221570109,-0.440860479379104,-0.496320182103172,0.559139462807474],[0,0,0,0],[8.999999E+09,8.999999E+09,8.999999E+09,8.999999E+09,8.999999E+09,8.999999E+09]];
	LOCAL CONST Robtarget Tr_meulage_bavure_P570 :=[[225.090390625,197.96328125,19.5],[0.496110936136754,-0.440271986990197,-0.496728579302687,0.559727822268244],[0,0,0,0],[8.999999E+09,8.999999E+09,8.999999E+09,8.999999E+09,8.999999E+09,8.999999E+09]];
	LOCAL CONST Robtarget Tr_meulage_bavure_P571 :=[[224.797296875,200.908875,19.5],[0.495448396013403,-0.439579721458981,-0.497223725397546,0.560418702642566],[0,0,0,0],[8.999999E+09,8.999999E+09,8.999999E+09,8.999999E+09,8.999999E+09,8.999999E+09]];
	LOCAL CONST Robtarget Tr_meulage_bavure_P572 :=[[224.68878125,201.8851875,19.5],[0.494652867720112,-0.438775313143973,-0.497822512861906,0.561219663518248],[0,0,0,0],[8.999999E+09,8.999999E+09,8.999999E+09,8.999999E+09,8.999999E+09,8.999999E+09]];
	LOCAL CONST Robtarget Tr_meulage_bavure_P573 :=[[224.57659375,203.904171875,19.5],[0.493654838470715,-0.437800936172737,-0.498579066470959,0.562186939743067],[0,0,0,0],[8.999999E+09,8.999999E+09,8.999999E+09,8.999999E+09,8.999999E+09,8.999999E+09]];
	LOCAL CONST Robtarget Tr_meulage_bavure_P574 :=[[224.078984375,209.4023125,19.5],[0.492410043766797,-0.436606982487831,-0.499523278537433,0.563367718137689],[0,0,0,0],[8.999999E+09,8.999999E+09,8.999999E+09,8.999999E+09,8.999999E+09,8.999999E+09]];
	LOCAL CONST Robtarget Tr_meulage_bavure_P575 :=[[224.03809375,209.886140625,19.5],[0.490868228924697,-0.435155645042599,-0.500692840518768,0.564796092296272],[0,0,0,0],[8.999999E+09,8.999999E+09,8.999999E+09,8.999999E+09,8.999999E+09,8.999999E+09]];
	LOCAL CONST Robtarget Tr_meulage_bavure_P576 :=[[223.33715625,216.5809375,19.5],[0.488983378832458,-0.433391859035336,-0.50211519760758,0.566521914915027],[0,0,0,0],[8.999999E+09,8.999999E+09,8.999999E+09,8.999999E+09,8.999999E+09,8.999999E+09]];
	LOCAL CONST Robtarget Tr_meulage_bavure_P577 :=[[223.075921875,221.04528125,19.5],[0.486712889428917,-0.431299490486626,-0.503822908010961,0.568554122430847],[0,0,0,0],[8.999999E+09,8.999999E+09,8.999999E+09,8.999999E+09,8.999999E+09,8.999999E+09]];
	LOCAL CONST Robtarget Tr_meulage_bavure_P578 :=[[222.850703125,224.7028125,19.5],[0.484026693482894,-0.428838265907807,-0.505827652222138,0.570924064947906],[0,0,0,0],[8.999999E+09,8.999999E+09,8.999999E+09,8.999999E+09,8.999999E+09,8.999999E+09]];
	LOCAL CONST Robtarget Tr_meulage_bavure_P579 :=[[222.6641875,226.612359375,19.5],[0.480908124386568,-0.425988299510064,-0.508131134053102,0.573641085684617],[0,0,0,0],[8.999999E+09,8.999999E+09,8.999999E+09,8.999999E+09,8.999999E+09,8.999999E+09]];
	LOCAL CONST Robtarget Tr_meulage_bavure_P580 :=[[222.077703125,232.0573125,19.5],[0.477342906879743,-0.422756333384185,-0.510738921492191,0.576685864148021],[0,0,0,0],[8.999999E+09,8.999999E+09,8.999999E+09,8.999999E+09,8.999999E+09,8.999999E+09]];
	LOCAL CONST Robtarget Tr_meulage_bavure_P581 :=[[221.856328125,233.539921875,19.5],[0.473342776896007,-0.419142460994193,-0.513627395170876,0.580045784298178],[0,0,0,0],[8.999999E+09,8.999999E+09,8.999999E+09,8.999999E+09,8.999999E+09,8.999999E+09]];
	LOCAL CONST Robtarget Tr_meulage_bavure_P582 :=[[221.63665625,234.732734375,19.5],[0.468913505015497,-0.415153139717017,-0.516780034219042,0.583700601018836],[0,0,0,0],[8.999999E+09,8.999999E+09,8.999999E+09,8.999999E+09,8.999999E+09,8.999999E+09]];
	LOCAL CONST Robtarget Tr_meulage_bavure_P583 :=[[220.549375,238.1279375,19.5],[0.464069501756382,-0.410802926087609,-0.520173873145089,0.587621983212574],[0,0,0,0],[8.999999E+09,8.999999E+09,8.999999E+09,8.999999E+09,8.999999E+09,8.999999E+09]];
	LOCAL CONST Robtarget Tr_meulage_bavure_P584 :=[[219.828921875,241.8514375,19.5],[0.458844015044118,-0.406110923299055,-0.523768456346992,0.591779259497383],[0,0,0,0],[8.999999E+09,8.999999E+09,8.999999E+09,8.999999E+09,8.999999E+09,8.999999E+09]];
	LOCAL CONST Robtarget Tr_meulage_bavure_P585 :=[[219.231203125,244.455203125,19.5],[0.453238799425272,-0.401094630789921,-0.527555408335533,0.596140066580803],[0,0,0,0],[8.999999E+09,8.999999E+09,8.999999E+09,8.999999E+09,8.999999E+09,8.999999E+09]];
	LOCAL CONST Robtarget Tr_meulage_bavure_P586 :=[[218.724859375,245.79578125,19.5],[0.447285075968181,-0.395767804828885,-0.531495239409947,0.600680211062115],[0,0,0,0],[8.999999E+09,8.999999E+09,8.999999E+09,8.999999E+09,8.999999E+09,8.999999E+09]];
	LOCAL CONST Robtarget Tr_meulage_bavure_P587 :=[[217.32415625,249.692625,19.5],[0.440978816159089,-0.390139262616269,-0.535583153537988,0.60537568922981],[0,0,0,0],[8.999999E+09,8.999999E+09,8.999999E+09,8.999999E+09,8.999999E+09,8.999999E+09]];
	LOCAL CONST Robtarget Tr_meulage_bavure_P588 :=[[216.898625,250.606625,19.5],[0.434327911213475,-0.384209590901103,-0.5397986421082,0.610212816793199],[0,0,0,0],[8.999999E+09,8.999999E+09,8.999999E+09,8.999999E+09,8.999999E+09,8.999999E+09]];
	LOCAL CONST Robtarget Tr_meulage_bavure_P589 :=[[216.628046875,251.475640625,19.5],[0.427324241653805,-0.377967867569019,-0.544132003940331,0.615186675626356],[0,0,0,0],[8.999999E+09,8.999999E+09,8.999999E+09,8.999999E+09,8.999999E+09,8.999999E+09]];
	LOCAL CONST Robtarget Tr_meulage_bavure_P590 :=[[215.491828125,253.919796875,19.5],[0.419956234338464,-0.371403045660966,-0.548576068588745,0.620290928424503],[0,0,0,0],[8.999999E+09,8.999999E+09,8.999999E+09,8.999999E+09,8.999999E+09,8.999999E+09]];
	LOCAL CONST Robtarget Tr_meulage_bavure_P591 :=[[214.857171875,255.641484375,19.5],[0.412188158400853,-0.364489721542919,-0.553140660310844,0.625526638021565],[0,0,0,0],[8.999999E+09,8.999999E+09,8.999999E+09,8.999999E+09,8.999999E+09,8.999999E+09]];
	LOCAL CONST Robtarget Tr_meulage_bavure_P592 :=[[214.409734375,256.6200625,19.5],[0.403995253164729,-0.357211777462699,-0.557827417576896,0.630885214331258],[0,0,0,0],[8.999999E+09,8.999999E+09,8.999999E+09,8.999999E+09,8.999999E+09,8.999999E+09]];
	LOCAL CONST Robtarget Tr_meulage_bavure_P593 :=[[214.0914375,257.40075,19.5],[0.395365971736272,-0.349544182950235,-0.562616716381667,0.636370209081629],[0,0,0,0],[8.999999E+09,8.999999E+09,8.999999E+09,8.999999E+09,8.999999E+09,8.999999E+09]];
	LOCAL CONST Robtarget Tr_meulage_bavure_P594 :=[[213.39703125,258.832765625,19.5],[0.386259524712045,-0.341465488043842,-0.567521044225705,0.641969441955901],[0,0,0,0],[8.999999E+09,8.999999E+09,8.999999E+09,8.999999E+09,8.999999E+09,8.999999E+09]];
	LOCAL CONST Robtarget Tr_meulage_bavure_P595 :=[[212.399046875,260.5024375,19.5],[0.376668103476596,-0.332960788247833,-0.572519073706293,0.647672883140258],[0,0,0,0],[8.999999E+09,8.999999E+09,8.999999E+09,8.999999E+09,8.999999E+09,8.999999E+09]];
	LOCAL CONST Robtarget Tr_meulage_bavure_P596 :=[[210.620359375,263.86065625,19.5],[0.366582159875886,-0.324020318623146,-0.577593298869941,0.653463338130475],[0,0,0,0],[8.999999E+09,8.999999E+09,8.999999E+09,8.999999E+09,8.999999E+09,8.999999E+09]];
	LOCAL CONST Robtarget Tr_meulage_bavure_P597 :=[[209.845890625,265.17328125,19.5],[0.356006027540317,-0.314643777596608,-0.582716154865498,0.659318499993341],[0,0,0,0],[8.999999E+09,8.999999E+09,8.999999E+09,8.999999E+09,8.999999E+09,8.999999E+09]];
	LOCAL CONST Robtarget Tr_meulage_bavure_P598 :=[[208.56915625,267.044625,19.5],[0.344949423750682,-0.304851709026606,-0.587870602748964,0.665194321218394],[0,0,0,0],[8.999999E+09,8.999999E+09,8.999999E+09,8.999999E+09,8.999999E+09,8.999999E+09]];
	LOCAL CONST Robtarget Tr_meulage_bavure_P599 :=[[206.85003125,269.19475,19.5],[0.333438961592916,-0.294654705601857,-0.593012645475261,0.67106859982043],[0,0,0,0],[8.999999E+09,8.999999E+09,8.999999E+09,8.999999E+09,8.999999E+09,8.999999E+09]];
	LOCAL CONST Robtarget Tr_meulage_bavure_P600 :=[[204.870234375,271.58784375,19.5],[0.321505560683923,-0.284094571087286,-0.598122105842571,0.676885806935332],[0,0,0,0],[8.999999E+09,8.999999E+09,8.999999E+09,8.999999E+09,8.999999E+09,8.999999E+09]];
	LOCAL CONST Robtarget Tr_meulage_bavure_P601 :=[[203.211734375,273.62146875,19.5],[0.309197063259898,-0.273208635109584,-0.603157837377011,0.682608849183557],[0,0,0,0],[8.999999E+09,8.999999E+09,8.999999E+09,8.999999E+09,8.999999E+09,8.999999E+09]];
	LOCAL CONST Robtarget Tr_meulage_bavure_P602 :=[[202.474734375,274.3179375,19.5],[0.296578645320671,-0.262045144526779,-0.608069734155567,0.688203928914732],[0,0,0,0],[8.999999E+09,8.999999E+09,8.999999E+09,8.999999E+09,8.999999E+09,8.999999E+09]];
	LOCAL CONST Robtarget Tr_meulage_bavure_P603 :=[[200.230828125,276.570875,19.5],[0.28368466247576,-0.250643058167034,-0.612842479679591,0.693631865450875],[0,0,0,0],[8.999999E+09,8.999999E+09,8.999999E+09,8.999999E+09,8.999999E+09,8.999999E+09]];
	LOCAL CONST Robtarget Tr_meulage_bavure_P604 :=[[196.11090625,280.58325,19.5],[0.270592020662065,-0.239064155929452,-0.617432675680703,0.698859913505938],[0,0,0,0],[8.999999E+09,8.999999E+09,8.999999E+09,8.999999E+09,8.999999E+09,8.999999E+09]];
	LOCAL CONST Robtarget Tr_meulage_bavure_P605 :=[[194.476078125,281.81340625,19.5],[0.257354014413142,-0.227355396845064,-0.621816515033015,0.70386266872385],[0,0,0,0],[8.999999E+09,8.999999E+09,8.999999E+09,8.999999E+09,8.999999E+09,8.999999E+09]];
	LOCAL CONST Robtarget Tr_meulage_bavure_P606 :=[[192.3773125,283.86378125,19.5],[0.244037075806742,-0.215583086120149,-0.625981367745572,0.708602262094886],[0,0,0,0],[8.999999E+09,8.999999E+09,8.999999E+09,8.999999E+09,8.999999E+09,8.999999E+09]];
	LOCAL CONST Robtarget Tr_meulage_bavure_P607 :=[[191.64825,284.3360625,19.5],[0.230688121098206,-0.203786872813815,-0.629913243551072,0.713066060650703],[0,0,0,0],[8.999999E+09,8.999999E+09,8.999999E+09,8.999999E+09,8.999999E+09,8.999999E+09]];
	LOCAL CONST Robtarget Tr_meulage_bavure_P608 :=[[191.2631875,284.60559375,19.5],[0.217364417843814,-0.192013971340357,-0.633595250151854,0.717245009498521],[0,0,0,0],[8.999999E+09,8.999999E+09,8.999999E+09,8.999999E+09,8.999999E+09,8.999999E+09]];
	LOCAL CONST Robtarget Tr_meulage_bavure_P609 :=[[186.3176875,287.8104375,19.5],[0.204116539020213,-0.180305918733792,-0.637014762248626,0.72113688495687],[0,0,0,0],[8.999999E+09,8.999999E+09,8.999999E+09,8.999999E+09,8.999999E+09,8.999999E+09]];
	LOCAL CONST Robtarget Tr_meulage_bavure_P610 :=[[181.7503125,290.356875,19.5],[0.190990681492424,-0.168708881045842,-0.640178505694839,0.724728469073516],[0,0,0,0],[8.999999E+09,8.999999E+09,8.999999E+09,8.999999E+09,8.999999E+09,8.999999E+09]];
	LOCAL CONST Robtarget Tr_meulage_bavure_P611 :=[[181.070375,290.71271875,19.5],[0.178029452521881,-0.157256424755229,-0.643079437903448,0.7280279990864],[0,0,0,0],[8.999999E+09,8.999999E+09,8.999999E+09,8.999999E+09,8.999999E+09,8.999999E+09]];
	LOCAL CONST Robtarget Tr_meulage_bavure_P612 :=[[176.239921875,292.84303125,19.5],[0.165261901311505,-0.145976033085724,-0.645726708258995,0.731037974376478],[0,0,0,0],[8.999999E+09,8.999999E+09,8.999999E+09,8.999999E+09,8.999999E+09,8.999999E+09]];
	LOCAL CONST Robtarget Tr_meulage_bavure_P613 :=[[175.836125,292.9968125,19.5],[0.15273450044965,-0.13491066881017,-0.648129210915734,0.733757323487361],[0,0,0,0],[8.999999E+09,8.999999E+09,8.999999E+09,8.999999E+09,8.999999E+09,8.999999E+09]];
	LOCAL CONST Robtarget Tr_meulage_bavure_P614 :=[[173.71253125,293.56525,19.5],[0.140478882155773,-0.124083528068876,-0.650283611045512,0.736206619731074],[0,0,0,0],[8.999999E+09,8.999999E+09,8.999999E+09,8.999999E+09,8.999999E+09,8.999999E+09]];
	LOCAL CONST Robtarget Tr_meulage_bavure_P615 :=[[171.76178125,294.26415625,19.5],[0.128526847142542,-0.113524000623468,-0.65220188798921,0.738394100835963],[0,0,0,0],[8.999999E+09,8.999999E+09,8.999999E+09,8.999999E+09,8.999999E+09,8.999999E+09]];
	LOCAL CONST Robtarget Tr_meulage_bavure_P616 :=[[169.792296875,294.68034375,19.5],[0.116911946736098,-0.103265045023597,-0.653905212708491,0.740321484207579],[0,0,0,0],[8.999999E+09,8.999999E+09,8.999999E+09,8.999999E+09,8.999999E+09,8.999999E+09]];
	LOCAL CONST Robtarget Tr_meulage_bavure_P617 :=[[166.344171875,295.74175,19.5],[0.105673436285712,-0.0933370319054641,-0.655390542863985,0.74201385409108],[0,0,0,0],[8.999999E+09,8.999999E+09,8.999999E+09,8.999999E+09,8.999999E+09,8.999999E+09]];
	LOCAL CONST Robtarget Tr_meulage_bavure_P618 :=[[165.0575,295.999875,19.5],[0.0948505478113717,-0.0837758894818504,-0.65667344714957,0.743481645859606],[0,0,0,0],[8.999999E+09,8.999999E+09,8.999999E+09,8.999999E+09,8.999999E+09,8.999999E+09]];
	LOCAL CONST Robtarget Tr_meulage_bavure_P619 :=[[162.405515625,296.73353125,19.5],[0.0844897958088553,-0.074625707387539,-0.657780422369321,0.7447263887823],[0,0,0,0],[8.999999E+09,8.999999E+09,8.999999E+09,8.999999E+09,8.999999E+09,8.999999E+09]];
	LOCAL CONST Robtarget Tr_meulage_bavure_P620 :=[[160.208,297.2576875,19.5],[0.0746447542840938,-0.065929031427793,-0.658703071517615,0.74578266743477],[0,0,0,0],[8.999999E+09,8.999999E+09,8.999999E+09,8.999999E+09,8.999999E+09,8.999999E+09]];
	LOCAL CONST Robtarget Tr_meulage_bavure_P621 :=[[157.466671875,297.60375,19.5],[0.0653604910524248,-0.0577279838412296,-0.659466973626058,0.746658420422284],[0,0,0,0],[8.999999E+09,8.999999E+09,8.999999E+09,8.999999E+09,8.999999E+09,8.999999E+09]];
	LOCAL CONST Robtarget Tr_meulage_bavure_P622 :=[[155.7241875,297.57721875,19.5],[0.0567129000336501,-0.050089695237385,-0.660087171148266,0.747368447210798],[0,0,0,0],[8.999999E+09,8.999999E+09,8.999999E+09,8.999999E+09,8.999999E+09,8.999999E+09]];
	LOCAL CONST Robtarget Tr_meulage_bavure_P623 :=[[152.557,297.85753125,19.5],[0.0487477705134357,-0.0430549541911881,-0.660584898333317,0.747928818727775],[0,0,0,0],[8.999999E+09,8.999999E+09,8.999999E+09,8.999999E+09,8.999999E+09,8.999999E+09]];
	LOCAL CONST Robtarget Tr_meulage_bavure_P624 :=[[151.84490625,297.84446875,19.5],[0.0415359340311119,-0.0366858313710959,-0.660974357644519,0.748359415319397],[0,0,0,0],[8.999999E+09,8.999999E+09,8.999999E+09,8.999999E+09,8.999999E+09,8.999999E+09]];
	LOCAL CONST Robtarget Tr_meulage_bavure_P625 :=[[150.590765625,297.91784375,19.5],[0.0351348406629365,-0.0310324957352833,-0.661267605984332,0.748683965672954],[0,0,0,0],[8.999999E+09,8.999999E+09,8.999999E+09,8.999999E+09,8.999999E+09,8.999999E+09]];
	LOCAL CONST Robtarget Tr_meulage_bavure_P626 :=[[146.5621875,297.88915625,19.5],[0.0296107749175343,-0.0261534844437419,-0.661479455467656,0.748921976746876],[0,0,0,0],[8.999999E+09,8.999999E+09,8.999999E+09,8.999999E+09,8.999999E+09,8.999999E+09]];
	LOCAL CONST Robtarget Tr_meulage_bavure_P627 :=[[142.615484375,298.0396875,19.5],[0.0250089654664302,-0.0220888240894529,-0.661625160618985,0.749091971878318],[0,0,0,0],[8.999999E+09,8.999999E+09,8.999999E+09,8.999999E+09,8.999999E+09,8.999999E+09]];
	LOCAL CONST Robtarget Tr_meulage_bavure_P628 :=[[142.072453125,297.98584375,19.5],[0.0213785625765336,-0.0188822767929466,-0.661723569345669,0.749205135098327],[0,0,0,0],[8.999999E+09,8.999999E+09,8.999999E+09,8.999999E+09,8.999999E+09,8.999999E+09]];
	LOCAL CONST Robtarget Tr_meulage_bavure_P629 :=[[141.47540625,297.98865625,19.5],[0.018759804451131,-0.016568883275829,-0.661776175662007,0.749283547911013],[0,0,0,0],[8.999999E+09,8.999999E+09,8.999999E+09,8.999999E+09,8.999999E+09,8.999999E+09]];
	LOCAL CONST Robtarget Tr_meulage_bavure_P630 :=[[137.7031875,297.56115625,19.5],[0.0171745868344647,-0.0151687268037614,-0.661807950641603,0.749323147755212],[0,0,0,0],[8.999999E+09,8.999999E+09,8.999999E+09,8.999999E+09,8.999999E+09,8.999999E+09]];
	LOCAL CONST Robtarget Tr_meulage_bavure_P631 :=[[135.226375,297.529,19.5],[0.0166477620892042,-0.0147035109416516,-0.661820468524339,0.749333254450671],[0,0,0,0],[8.999999E+09,8.999999E+09,8.999999E+09,8.999999E+09,8.999999E+09,8.999999E+09]];
	LOCAL CONST Robtarget Tr_meulage_bavure_degg1 :=[[135.66708818823,307.442586099788,18.2644505158357],[0.0166477620892042,-0.0147035109416516,-0.661820468524339,0.749333254450671],[0,0,0,0],[8.999999E+09,8.999999E+09,8.999999E+09,8.999999E+09,8.999999E+09,8.999999E+09]];
	LOCAL CONST Robtarget Tr_meulage_bavure_degg2 :=[[144.040638764607,495.800721995751,-5.21098968328505],[0.0166477620892042,-0.0147035109416516,-0.661820468524339,0.749333254450671],[0,0,0,0],[8.999999E+09,8.999999E+09,8.999999E+09,8.999999E+09,8.999999E+09,8.999999E+09]];
	LOCAL PROC Tr_pick()
		!!Programme Tr_pick - 04/04/2023 12:19:29;
		 CONST Robtarget Ppick :=[[-47.1877218952358,17.5876932064478,41.9822435148333],[-0.00295481298502662,0.783175650666835,-0.621786151399891,0.00302509671164741],[0,0,0,0],[8.999999E+09,8.999999E+09,8.999999E+09,8.999999E+09,8.999999E+09,8.999999E+09]];
		 VAR Pose Ref :=[[0,0,0],[1,0,0,0]];
		LocalisationPieceTable 106 \model:=0;
		MoveJ Reltool(Ppick,0,0,-200),V1000,Z0,Tool_Prehenseur \Wobj:=Wobj_vision;
		MoveL Reltool(Ppick,0,0,-100),V500,Z0,Tool_Prehenseur \Wobj:=Wobj_vision;
		MoveL Reltool(Ppick,0,0,-10),V200,Z0,Tool_Prehenseur \Wobj:=Wobj_vision;
		MoveL Ppick,V100,Fine,Tool_Prehenseur \Wobj:=Wobj_vision;
		Gripper_Close;
		MoveL Reltool(Ppick,0,0,-200),V500,Z0,Tool_Prehenseur \Wobj:=Wobj_vision;
		LocalisationPiecePrehenseur 106 \model:=0,Ref;
	ENDPROC
	LOCAL PROC Tr_Cut()
		!!Programme Tr_Cut - 04/04/2023 12:19:29;
		confJ \off;
		confL \off;
		Tool := ToolOffset(Tool_M2_D490_S180);
		MoveAbsJ [[0,-40,40,0,90,0],[8.999999E+09,8.999999E+09,8.999999E+09,8.999999E+09,8.999999E+09,8.999999E+09]] ,V1000,Z0,Tool_M2_D490_S180 \Wobj:=Wobj_Part_0;
		Movej Reltool(Coupe_0,-200,0,-20.9771796875),V1000,Z0,Tool_M2_D490_S180 \Wobj:=Wobj_Part_0;
		MoveL Reltool(Coupe_0,0,0,-20.9771796875),V500,Z0,Tool_M2_D490_S180 \Wobj:=Wobj_Part_0;
		MoveL Reltool(Coupe_0,0,0,-10.9771796875),vitesse_Tronconnage,Z0,Tool_M2_D490_S180 \Wobj:=Wobj_Part_0;
		MoveL Coupe_0,vitesse_Tronconnage,Fine,Tool_M2_D490_S180 \Wobj:=Wobj_Part_0;
		MoveL Reltool(Coupe_0,0,0,10.9771796875),vitesse_Tronconnage,Z0,Tool_M2_D490_S180 \Wobj:=Wobj_Part_0;
		MoveL Reltool(Coupe_0,-200,0,10.9771796875),V500,Z0,Tool_M2_D490_S180 \Wobj:=Wobj_Part_0;
	ENDPROC
	LOCAL PROC Tr_meulage_motif_1()
		!!Programme Tr_meulage_motif_1 - 04/04/2023 12:19:29;
		 CONST Speeddata vitesse_Meulage :=[50, 500, 0, 0];
		confJ \off;
		confL \off;
		Tool := ToolOffset(Tool_M1_D500_S0);
		MoveAbsJ [[0,-40,40,0,90,0],[8.999999E+09,8.999999E+09,8.999999E+09,8.999999E+09,8.999999E+09,8.999999E+09]] ,V1000,Z0,Tool_M1_D500_S0 \Wobj:=Wobj_Part_0;
		MoveJ Tr_meulage_motif_1_App1,V2000,Z100,Tool,\Wobj:=Wobj_Part_0;
		MoveJ Tr_meulage_motif_1_App2,V500,Z0,Tool,\Wobj:=Wobj_Part_0;
		MoveL Tr_meulage_motif_1_P0,[12.5,500,0,0],z0,Tool \wobj:=Wobj_Part_0;
		MoveL Tr_meulage_motif_1_P1,[12.5,500,0,0],z0,Tool \wobj:=Wobj_Part_0;
		MoveL Tr_meulage_motif_1_P2,[12.5,500,0,0],z0,Tool \wobj:=Wobj_Part_0;
		MoveL Tr_meulage_motif_1_P3,[12.5,500,0,0],z0,Tool \wobj:=Wobj_Part_0;
		MoveL Tr_meulage_motif_1_P4,[12.5,500,0,0],z0,Tool \wobj:=Wobj_Part_0;
		MoveL Tr_meulage_motif_1_P5,[12.5,500,0,0],z0,Tool \wobj:=Wobj_Part_0;
		MoveL Tr_meulage_motif_1_P6,[12.5,500,0,0],z0,Tool \wobj:=Wobj_Part_0;
		MoveL Tr_meulage_motif_1_P7,[12.5,500,0,0],z0,Tool \wobj:=Wobj_Part_0;
		MoveL Tr_meulage_motif_1_P8,[12.5,500,0,0],z0,Tool \wobj:=Wobj_Part_0;
		MoveL Tr_meulage_motif_1_P9,[12.5,500,0,0],z0,Tool \wobj:=Wobj_Part_0;
		MoveL Tr_meulage_motif_1_P10,[12.5,500,0,0],z0,Tool \wobj:=Wobj_Part_0;
		MoveL Tr_meulage_motif_1_P11,[12.5,500,0,0],z0,Tool \wobj:=Wobj_Part_0;
		MoveL Tr_meulage_motif_1_P12,[12.5,500,0,0],z0,Tool \wobj:=Wobj_Part_0;
		MoveL Tr_meulage_motif_1_P13,[12.5,500,0,0],z0,Tool \wobj:=Wobj_Part_0;
		MoveL Tr_meulage_motif_1_P14,[12.5,500,0,0],z0,Tool \wobj:=Wobj_Part_0;
		MoveL Tr_meulage_motif_1_P15,[12.5,500,0,0],z0,Tool \wobj:=Wobj_Part_0;
		MoveL Tr_meulage_motif_1_P16,[12.5,500,0,0],z0,Tool \wobj:=Wobj_Part_0;
		MoveL Tr_meulage_motif_1_P17,[12.5,500,0,0],z0,Tool \wobj:=Wobj_Part_0;
		MoveL Tr_meulage_motif_1_P18,[12.5,500,0,0],z0,Tool \wobj:=Wobj_Part_0;
		MoveL Tr_meulage_motif_1_P19,[12.5,500,0,0],z0,Tool \wobj:=Wobj_Part_0;
		MoveL Tr_meulage_motif_1_P20,[12.5,500,0,0],z0,Tool \wobj:=Wobj_Part_0;
		MoveL Tr_meulage_motif_1_P21,[12.5,500,0,0],z0,Tool \wobj:=Wobj_Part_0;
		MoveL Tr_meulage_motif_1_P22,[12.5,500,0,0],z0,Tool \wobj:=Wobj_Part_0;
		MoveL Tr_meulage_motif_1_P23,[12.5,500,0,0],z0,Tool \wobj:=Wobj_Part_0;
		MoveL Tr_meulage_motif_1_P24,[12.5,500,0,0],z0,Tool \wobj:=Wobj_Part_0;
		MoveL Tr_meulage_motif_1_P25,[12.5,500,0,0],z0,Tool \wobj:=Wobj_Part_0;
		MoveL Tr_meulage_motif_1_P26,[12.5,500,0,0],z0,Tool \wobj:=Wobj_Part_0;
		MoveL Tr_meulage_motif_1_P27,[12.5,500,0,0],z0,Tool \wobj:=Wobj_Part_0;
		MoveL Tr_meulage_motif_1_P28,[12.5,500,0,0],z0,Tool \wobj:=Wobj_Part_0;
		MoveL Tr_meulage_motif_1_P29,[12.5,500,0,0],z0,Tool \wobj:=Wobj_Part_0;
		MoveL Tr_meulage_motif_1_P30,[12.5,500,0,0],z0,Tool \wobj:=Wobj_Part_0;
		MoveL Tr_meulage_motif_1_P31,[12.5,500,0,0],z0,Tool \wobj:=Wobj_Part_0;
		MoveL Tr_meulage_motif_1_P32,[12.5,500,0,0],z0,Tool \wobj:=Wobj_Part_0;
		MoveL Tr_meulage_motif_1_P33,[12.5,500,0,0],z0,Tool \wobj:=Wobj_Part_0;
		MoveL Tr_meulage_motif_1_P34,[12.5,500,0,0],z0,Tool \wobj:=Wobj_Part_0;
		MoveL Tr_meulage_motif_1_P35,[12.5,500,0,0],z0,Tool \wobj:=Wobj_Part_0;
		MoveL Tr_meulage_motif_1_P36,[12.5,500,0,0],z0,Tool \wobj:=Wobj_Part_0;
		MoveL Tr_meulage_motif_1_P37,[12.5,500,0,0],z0,Tool \wobj:=Wobj_Part_0;
		MoveL Tr_meulage_motif_1_P38,[12.5,500,0,0],z0,Tool \wobj:=Wobj_Part_0;
		MoveL Tr_meulage_motif_1_P39,[12.5,500,0,0],z0,Tool \wobj:=Wobj_Part_0;
		MoveL Tr_meulage_motif_1_P40,[12.5,500,0,0],z0,Tool \wobj:=Wobj_Part_0;
		MoveL Tr_meulage_motif_1_P41,[12.5,500,0,0],z0,Tool \wobj:=Wobj_Part_0;
		MoveL Tr_meulage_motif_1_P42,[12.5,500,0,0],z0,Tool \wobj:=Wobj_Part_0;
		MoveL Tr_meulage_motif_1_P43,[12.5,500,0,0],z0,Tool \wobj:=Wobj_Part_0;
		MoveL Tr_meulage_motif_1_P44,[12.5,500,0,0],z0,Tool \wobj:=Wobj_Part_0;
		MoveL Tr_meulage_motif_1_P45,[12.5,500,0,0],z0,Tool \wobj:=Wobj_Part_0;
		MoveL Tr_meulage_motif_1_P46,[12.5,500,0,0],z0,Tool \wobj:=Wobj_Part_0;
		MoveL Tr_meulage_motif_1_P47,[12.5,500,0,0],z0,Tool \wobj:=Wobj_Part_0;
		MoveL Tr_meulage_motif_1_P48,[12.5,500,0,0],z0,Tool \wobj:=Wobj_Part_0;
		MoveL Tr_meulage_motif_1_P49,[12.5,500,0,0],z0,Tool \wobj:=Wobj_Part_0;
		MoveL Tr_meulage_motif_1_P50,[12.5,500,0,0],z0,Tool \wobj:=Wobj_Part_0;
		MoveL Tr_meulage_motif_1_P51,[12.5,500,0,0],z0,Tool \wobj:=Wobj_Part_0;
		MoveL Tr_meulage_motif_1_P52,[12.5,500,0,0],z0,Tool \wobj:=Wobj_Part_0;
		MoveL Tr_meulage_motif_1_P53,[12.5,500,0,0],z0,Tool \wobj:=Wobj_Part_0;
		MoveL Tr_meulage_motif_1_P54,[12.5,500,0,0],z0,Tool \wobj:=Wobj_Part_0;
		MoveL Tr_meulage_motif_1_P55,[12.5,500,0,0],z0,Tool \wobj:=Wobj_Part_0;
		MoveL Tr_meulage_motif_1_P56,[12.5,500,0,0],z0,Tool \wobj:=Wobj_Part_0;
		MoveL Tr_meulage_motif_1_P57,[12.5,500,0,0],z0,Tool \wobj:=Wobj_Part_0;
		MoveL Tr_meulage_motif_1_P58,[12.5,500,0,0],z0,Tool \wobj:=Wobj_Part_0;
		MoveL Tr_meulage_motif_1_P59,[12.5,500,0,0],z0,Tool \wobj:=Wobj_Part_0;
		MoveL Tr_meulage_motif_1_P60,[12.5,500,0,0],z0,Tool \wobj:=Wobj_Part_0;
		MoveL Tr_meulage_motif_1_P61,[12.5,500,0,0],z0,Tool \wobj:=Wobj_Part_0;
		MoveL Tr_meulage_motif_1_P62,[12.5,500,0,0],z0,Tool \wobj:=Wobj_Part_0;
		MoveL Tr_meulage_motif_1_P63,[12.5,500,0,0],z0,Tool \wobj:=Wobj_Part_0;
		MoveL Tr_meulage_motif_1_P64,[12.5,500,0,0],z0,Tool \wobj:=Wobj_Part_0;
		MoveL Tr_meulage_motif_1_P65,[12.5,500,0,0],z0,Tool \wobj:=Wobj_Part_0;
		MoveL Tr_meulage_motif_1_P66,[12.5,500,0,0],z0,Tool \wobj:=Wobj_Part_0;
		MoveL Tr_meulage_motif_1_P67,[12.5,500,0,0],z0,Tool \wobj:=Wobj_Part_0;
		MoveL Tr_meulage_motif_1_P68,[12.5,500,0,0],z0,Tool \wobj:=Wobj_Part_0;
		MoveL Tr_meulage_motif_1_P69,[12.5,500,0,0],z0,Tool \wobj:=Wobj_Part_0;
		MoveL Tr_meulage_motif_1_P70,[12.5,500,0,0],z0,Tool \wobj:=Wobj_Part_0;
		MoveL Tr_meulage_motif_1_P71,[12.5,500,0,0],z0,Tool \wobj:=Wobj_Part_0;
		MoveL Tr_meulage_motif_1_P72,[12.5,500,0,0],z0,Tool \wobj:=Wobj_Part_0;
		MoveL Tr_meulage_motif_1_P73,[12.5,500,0,0],z0,Tool \wobj:=Wobj_Part_0;
		MoveL Tr_meulage_motif_1_P74,[12.5,500,0,0],z0,Tool \wobj:=Wobj_Part_0;
		MoveL Tr_meulage_motif_1_P75,[12.5,500,0,0],z0,Tool \wobj:=Wobj_Part_0;
		MoveL Tr_meulage_motif_1_P76,[12.5,500,0,0],z0,Tool \wobj:=Wobj_Part_0;
		MoveL Tr_meulage_motif_1_P77,[12.5,500,0,0],z0,Tool \wobj:=Wobj_Part_0;
